// TwinCAT 3 PLC project Main
// ProgramVersion: 3.1.4024.0
// libraries:
//   Tc2_Standard, * (Beckhoff Automation GmbH)
//   Tc2_System, * (Beckhoff Automation GmbH)
//   Tc2_Utilities, * (Beckhoff Automation GmbH)
//   Tc3_DynamicMemory, * (Beckhoff Automation GmbH)
//   Tc3_JsonXml, * (Beckhoff Automation GmbH)
//   Tc3_Module, * (Beckhoff Automation GmbH)
//   TcUnit, * (www.tcunit.org)
//   mobject-core,0.4.0,mobject
// project tree:
//   mobject-collections/ MobjectCollectionsExample.TcPOU, MobjectCollectionsUnitTests.TcPOU
//   mobject-collections/Tests/ DictionaryForwardEnumerator_TestSuite.TcPOU (not stored), DictionaryKeyValueForwardEnumerator_TestSuite.TcPOU, Dictionary_TestSuite.TcPOU, LinkedListForwardEnumerator_TestSuite.TcPOU (not stored), LinkedList_TestSuite.TcPOU (not stored), OrderedDicKeyValueForwardEnumerator_TestSuite.TcPOU (not stored), OrderedDictionaryForwardEnumerator_TestSuite.TcPOU, OrderedDictionary_TestSuite.TcPOU, QueueForwardEnumerator_TestSuite.TcPOU (not stored), Queue_TestSuite.TcPOU, StackForwardEnumerator_TestSuite.TcPOU, Stack_TestSuite.TcPOU (not stored)
//   mobject-collections/Tests/Mocks/EventHandlers/ CollectionChangedEventHandler.TcPOU (not stored), CollectionDisposedEventHandler.TcPOU, CollectionEventHandler.TcPOU, CollectionEventHandlerBase.TcPOU (not stored), KeyValueCollectionChangedEventHandler.TcPOU, KeyValueCollectionDisposedEventHandler.TcPOU (not stored), KeyValueCollectionEventHandler.TcPOU (not stored)
//   mobject-converters/ MobjectConvertersUnitTests.TcPOU (not stored)
//   mobject-converters/Tests/ BOOL_TO_TestSuite.TcPOU, BYTE_TO_TestSuite.TcPOU (not stored), DATE_TO_TestSuite.TcPOU (not stored), DINT_TO_TestSuite.TcPOU (not stored), DT_TO_TestSuite.TcPOU, DWORD_TO_TestSuite.TcPOU, INT_TO_TestSuite.TcPOU (not stored), LINT_TO_TestSuite.TcPOU (not stored), LREAL_TO_TestSuite.TcPOU (not stored), LWORD_TO_TestSuite.TcPOU (not stored), REAL_TO_TestSuite.TcPOU (not stored), SINT_TO_TestSuite.TcPOU, STRING_TO_TestSuite.TcPOU (not stored), TIME_TO_TestSuite.TcPOU (not stored), TOD_TO_TestSuite.TcPOU (not stored), UDINT_TO_TestSuite.TcPOU (not stored), UINT_TO_TestSuite.TcPOU, ULINT_TO_TestSuite.TcPOU (not stored), USINT_TO_TestSuite.TcPOU (not stored), WORD_TO_TestSuite.TcPOU
//   mobject-datatypes/ MobjectDatatypesUnitTests.TcPOU
//   mobject-datatypes/Tests/ AliasDatatype_TestSuite.TcPOU, Datatype_TestSuite.TcPOU, EnumDatatype_TestSuite.TcPOU (not stored), StructuredDatatype_TestSuite.TcPOU, _ArrayDatatype_1D_TestSuite.TcPOU (not stored), _ArrayDatatype_2D_TestSuite.TcPOU, _ArrayDatatype_3D_TestSuite.TcPOU (not stored), _BIT_UsingMockStructure_TestSuite.TcPOU (not stored), _BOOL_TestSuite.TcPOU, _BYTE_TestSuite.TcPOU, _DINT_TestSuite.TcPOU (not stored), _DT_TestSuite.TcPOU, _DWORD_TestSuite.TcPOU, _INT_TestSuite.TcPOU, _LINT_TestSuite.TcPOU (not stored), _LREAL_TestSuite.TcPOU, _LWORD_TestSuite.TcPOU, _REAL_TestSuite.TcPOU (not stored), _SINT_TestSuite.TcPOU (not stored), _STRING_TestSuite.TcPOU, _TIME_OF_DAY_TestSuite.TcPOU, _TOD_TestSuite.TcPOU, _UDINT_TestSuite.TcPOU (not stored), _UINT_TestSuite.TcPOU (not stored), _ULINT_TestSuite.TcPOU (not stored), _USINT_TestSuite.TcPOU, _WORD_TestSuite.TcPOU
//   mobject-datatypes/Tests/Mocks/1DimArray/ _Array0to10OfBool.TcPOU
//   mobject-datatypes/Tests/Mocks/2DimArray/ _Array0to1_0to2OfBool.TcPOU
//   mobject-datatypes/Tests/Mocks/3DimArray/ _Array0to1_0to2_0to3OfBool.TcPOU
//   mobject-datatypes/Tests/Mocks/DUT/ MyStruct.TcDUT (not stored)
//   mobject-datatypes/Tests/Mocks/ MockAliasDatatype_HRESULT.TcPOU, MockDatatype_BOOL.TcPOU, MockEnumDatatype_E_TcEventClass.TcPOU, MockStructuredDatatype_TIMESTRUCT.TcPOU, _MyStruct.TcPOU
//   mobject-deserialization/ MobjectDeserializationUnitTests.TcPOU
//   mobject-deserialization/Tests/ CustomDeserializationFailedError_TestSuite.TcPOU (not stored), DeserializationErrorFactory_TestSuite.TcPOU (not stored), DeserializerGarbageCollector_TestSuite.TcPOU, IncorrectKeyTypeDeserializationError_TestSuite.TcPOU (not stored), IncorrectTypeDeserializationError_TestSuite.TcPOU (not stored), InvalidKeyDeserializationError_TestSuite.TcPOU (not stored), MissingKeyDeserializationError_TestSuite.TcPOU, InvalidArrayIndexDeserializationError_TestSuite.TcPOU
//   mobject-deserialization/Tests/Mocks/ MockDisposableDeserializer.TcPOU
//   mobject-disposable/ MobjectDisposableUnitTests.TcPOU (not stored)
//   mobject-disposable/Tests/ Disposable_TestSuite.TcPOU (not stored)
//   mobject-disposable/Tests/Mocks/ MockDisposable.TcPOU (not stored)
//   mobject-errors/ MobjectErrorsUnitTests.TcPOU (not stored)
//   mobject-errors/Tests/ Error_TestSuite.TcPOU, NullError_TestSuite.TcPOU
//   mobject-events/ MobjectEventsUnitTests.TcPOU (not stored)
//   mobject-events/Tests/ EventEmitterInterface_TestSuite.TcPOU, EventEmitter_TestSuite.TcPOU, EventHandlerInterface_TestSuite.TcPOU, EventTargetInterface_TestSuite.TcPOU (not stored)
//   mobject-events/Tests/Mocks/ MockEvent.TcPOU, MockEventHandler.TcPOU
//   mobject-json/ MobjectJsonUnitTests.TcPOU (not stored)
//   mobject-json/Tests/ JsonDeserializerArrayForwardEnumerator_TestSuite.TcPOU (not stored), JsonDeserializerObjectForwardEnumerator_TestSuite.TcPOU, JsonDeserializer_TestSuite.TcPOU, JsonDomParser_TestSuite.TcPOU (not stored), JsonSerializer_TestSuite.TcPOU
//   mobject-json/Tests/Mocks/ MockDeserializableUserObject.TcPOU (not stored), MockSerializableArray.TcPOU, MockSerializableUserObject.TcPOU (not stored)
//   / PlcTask.TcTTO (not stored)
//   Main/ MAIN.TcPOU
//   SharedMocks/ MockError.TcPOU (not stored), MockErrorVisitor.TcPOU, MockJsonSerializer.TcPOU (not stored)
// real-time tasks:
//   TASK PlcTask: cycle T#10ms, priority 20, ADS port 350

// ---- mobject-collections/MobjectCollectionsExample.TcPOU
PROGRAM MobjectCollectionsExample
VAR
END_VAR

END_PROGRAM

// ---- mobject-collections/MobjectCollectionsUnitTests.TcPOU
PROGRAM MobjectCollectionsUnitTests
VAR
	dictionary_TestSuite : Dictionary_TestSuite;
	dictionaryForwardEnumerator_TestSuite : DictionaryForwardEnumerator_TestSuite;
	dictionaryKeyValueForwardEnumerator_TestSuite : DictionaryKeyValueForwardEnumerator_TestSuite;
	orderedDictionary_TestSuite : OrderedDictionary_TestSuite;
	orderedDictionaryForwardEnumerator_TestSuite : OrderedDictionaryForwardEnumerator_TestSuite;
	orderedDicKeyValueForwardEnumerator_TestSuite : OrderedDicKeyValueForwardEnumerator_TestSuite;
    linkedList_TestSuite : LinkedList_TestSuite;
	linkedListForwardEnumerator_TestSuite : LinkedListForwardEnumerator_TestSuite;
    list_TestSuite : List_TestSuite;
    listEnumerator_TestSuite : ListForwardEnumerator_TestSuite;
	queue_TestSuite : Queue_TestSuite;
	queueForwardEnumerator_TestSuite : QueueForwardEnumerator_TestSuite;
    stack_TestSuite : Stack_TestSuite;
	stackForwardEnumerator_TestSuite : StackForwardEnumerator_TestSuite;
END_VAR

END_PROGRAM

// ---- mobject-collections/Tests/Dictionary_TestSuite.TcPOU
FUNCTION_BLOCK Dictionary_TestSuite EXTENDS TcUnit.FB_TestSuite
VAR
END_VAR

CheckAddOrUpdateCorrectlyAddsNewKey();
CheckAddOrUpdateCorrectlyUpdatesExistingKey();
CheckClear();
CheckContainsKeyIsFalse();
CheckContainsKeyIsTrue();
CheckCount();
CheckEnumeratorIsInvalidAfterChange();
CheckGetEnumerator();
CheckGetKeysReturnsACollection();
CheckGetKeysReturnsACollectionOfValidKeys();
CheckOffEvent();
CheckOnceEvent();
CheckOnChangedEvent();
CheckOnDisposedEvent();
CheckRemoveExisting();
CheckRemoveNonExisting();
CheckTryAddCorrectlyAddsNewKey();
CheckTryAddCorrectlyIgnoresUpdateWhenDuplicateFound();
CheckTryAddCorrectlyReturnsFalseWhenDuplicateFound();
CheckTryAddCorrectlyReturnsTrueWhenAddNewKey();
CheckTryGetValueTo();
CheckTryGetValue();
CheckWorksWithArrays();
CheckWorksWithIntegers();
CheckWorksWithStrings();
CheckIsEmptyWhenEmpty();
CheckIsEmptyWhenFull();

METHOD PUBLIC CheckAddOrUpdateCorrectlyAddsNewKey
VAR
	in : INT := 123;
	out : INT;
	expected : INT := 123;
	dictionary : Dictionary;
END_VAR
TEST('CheckAddOrUpdateCorrectlyAddsNewKey');

dictionary.AddOrUpdate('a',in);
dictionary.TryGetValue('a',out);

AssertEquals(
	Expected := expected,
	Actual := out,
	Message := 'Did not produce the expected result'
);

TEST_FINISHED();
END_METHOD

METHOD PUBLIC CheckAddOrUpdateCorrectlyUpdatesExistingKey
VAR
	in1 : INT := 123;
	in2 : INT := 456;
	out : INT;
	expected : INT := 456;
	dictionary : Dictionary;
END_VAR
TEST('CheckAddOrUpdateCorrectlyUpdatesExistingKey');

dictionary.AddOrUpdate('a',in1);
dictionary.AddOrUpdate('a',in2);
dictionary.TryGetValue('a',out);

AssertEquals(
	Expected := expected,
	Actual := out,
	Message := 'Did not produce the expected result'
);

TEST_FINISHED();
END_METHOD

METHOD PUBLIC CheckClear
VAR
	in1 : INT := 123;
	in2 : INT := 456;
	out : INT;
	expected : INT := 456;
	dictionary : Dictionary;
END_VAR
TEST('CheckClear');

dictionary.TryAdd('a',in1);
dictionary.Clear();
dictionary.TryAdd('a',in2); // if the dictionary was not empty then this would fail.
dictionary.TryGetValue('a',out);

// @TEST-ASSSERT
AssertEquals(
	Expected := expected,
	Actual := out,
	Message := 'Did not produce the expected result'
);

TEST_FINISHED();
END_METHOD

METHOD PUBLIC CheckContainsKeyIsFalse
VAR
	in1 : INT := 123;
	in2 : INT := 456;
	in3 : INT := 789;
	result : BOOL;
	dictionary : Dictionary;
END_VAR
TEST('CheckContainsKeyIsFalse');

dictionary.TryAdd('a',in1);
dictionary.TryAdd('b',in2);
dictionary.TryAdd('c',in3);

result := dictionary.ContainsKey('d');

AssertFalse(
	Condition := result,
	Message := 'Did not produce the expected result'
);

TEST_FINISHED();
END_METHOD

METHOD PUBLIC CheckContainsKeyIsTrue
VAR
	in1 : INT := 123;
	in2 : INT := 456;
	in3 : INT := 789;
	result : BOOL;
	dictionary : Dictionary;
END_VAR
TEST('CheckContainsKeyIsTrue');

dictionary.TryAdd('a',in1);
dictionary.TryAdd('b',in2);
dictionary.TryAdd('c',in3);

result := dictionary.ContainsKey('b');

AssertTrue(
	Condition := result,
	Message := 'Did not produce the expected result'
);

TEST_FINISHED();
END_METHOD

METHOD PUBLIC CheckCount
VAR
	in1 : INT := 123;
	in2 : INT := 456;
	in3 : INT := 789;
	out : DINT;
	expected : DINT := 3;
	dictionary : Dictionary;
END_VAR
TEST('CheckCount');

dictionary.TryAdd('a',in1);
dictionary.TryAdd('b',in2);
dictionary.TryAdd('c',in3);
out := dictionary.Count;

AssertEquals(
	Expected := expected,
	Actual := out,
	Message := 'Did not produce the expected result'
);

TEST_FINISHED();
END_METHOD

METHOD PUBLIC CheckEnumeratorIsInvalidAfterChange
VAR
	in : INT := 123;
	result : BOOL;
	dictionary : Dictionary;
	enumerator : I_ForwardEnumerator;
END_VAR
TEST('CheckEnumeratorIsInvalidAfterChange');

enumerator := dictionary.GetEnumerator();
dictionary.TryAdd('a',in);

result := enumerator.IsValid;
enumerator.Dispose();

AssertFalse(
	Condition := result,
	Message := 'Method returned true'
);

TEST_FINISHED();
END_METHOD

METHOD PUBLIC CheckGetEnumerator
VAR
	enumerator : I_ForwardEnumerator;
	dictionary : Dictionary;
END_VAR
TEST('CheckGetEnumerator');

enumerator := dictionary.GetEnumerator();

AssertTrue(
	Condition := (enumerator <> 0),
	Message := 'Did not return an enumerator'
);

enumerator.Dispose();

TEST_FINISHED();
END_METHOD

METHOD PUBLIC CheckGetKeysReturnsACollection
VAR
	result : BOOL;
	dictionary : Dictionary;
	collection : I_Collection;
END_VAR
TEST('CheckGetKeysReturnsACollection');

collection := dictionary.GetKeys();

result := collection <> 0;

IF result THEN
	collection.Dispose();
END_IF

AssertTrue(
	Condition := result,
	Message := 'Did not produce the expected result'
);

TEST_FINISHED();
END_METHOD

METHOD PUBLIC CheckGetKeysReturnsACollectionOfValidKeys
VAR
	in1 : INT := 123;
	in2 : INT := 456;
	in3 : INT := 789;
	out : ARRAY [0..2] OF T_MAXSTRING;
	expected : ARRAY [0..2] OF T_MAXSTRING;
	result,resulta,resultb,resultc : BOOL;
	dictionary : Dictionary;
	collection : I_Collection;
END_VAR
TEST('CheckGetKeysReturnsACollectionOfValidKeys');

// clear the out and expected variables as strings may contain left over data
memset(ADR(out),0,SIZEOF(out));
memset(ADR(expected),0,SIZEOF(expected));

// now create the "expected"
expected[0] := 'a';
expected[1] := 'b';
expected[2] := 'c';

// now setup the test
dictionary.TryAdd('a',in1);
dictionary.TryAdd('b',in2);
dictionary.TryAdd('c',in3);

collection := dictionary.GetKeys();
collection.TryCopyTo(out);
collection.Dispose();

// create the test result
resulta := expected[0] = out[0];
resultb := expected[1] = out[1];
resultc := expected[2] = out[2];
result := resulta AND resultb AND resultc;

AssertTrue(
	Condition := result,
	Message := 'Did not return an enumerator'
);

TEST_FINISHED();
END_METHOD

METHOD PUBLIC CheckIsEmptyWhenEmpty
VAR
	result : BOOL;
	dictionary : Dictionary;
END_VAR
TEST('CheckIsEmptyWhenEmpty');

// @TEST-RUN
result := dictionary.IsEmpty;

// @TEST-ASSSERT
AssertTrue(
	Condition := result,
	Message := 'Incorrect state of IsEmpty'
);

TEST_FINISHED();
END_METHOD

METHOD PUBLIC CheckIsEmptyWhenFull
VAR
	in : INT := 123;
	result : BOOL;
	dictionary : Dictionary;
END_VAR
TEST('CheckIsEmptyWhenFull');

// @TEST-FIXTURE
dictionary.AddOrUpdate('a',in);

// @TEST-RUN
result := dictionary.IsEmpty;

// @TEST-ASSSERT
AssertFalse(
	Condition := result,
	Message := 'Incorrect state of IsEmpty'
);

TEST_FINISHED();
END_METHOD

METHOD PUBLIC CheckOffEvent
VAR
	value : INT := 123;
	dictionary : Dictionary;
	handler : KeyValueCollectionChangedEventHandler(ExpectedOriginator := dictionary);
END_VAR
TEST('CheckOffEvent');

dictionary.OnEvent('OnChanged',handler);
dictionary.OffEvent('OnChanged',handler);

dictionary.TryAdd('a',value);

AssertFalse(
	Condition := handler.EventReceived,
	Message := 'OnceEvent emitted the OnChanged event more than once'
);

TEST_FINISHED();
END_METHOD

METHOD PUBLIC CheckOnceEvent
VAR
	value : INT := 123;
	dictionary : Dictionary;
	handler : KeyValueCollectionChangedEventHandler(ExpectedOriginator := dictionary);
END_VAR
TEST('CheckOnceEvent');

dictionary.OnceEvent('OnChanged',handler);
dictionary.TryAdd('a',value);
handler.Reset();

dictionary.TryAdd('a',value);

AssertFalse(
	Condition := handler.EventReceived,
	Message := 'OnceEvent emitted the OnChanged event more than once'
);

TEST_FINISHED();
END_METHOD

METHOD PUBLIC CheckOnChangedEvent
VAR
	value : INT := 123;
	dictionary : Dictionary;
	handler : KeyValueCollectionChangedEventHandler(ExpectedOriginator := dictionary);
END_VAR
TEST('CheckOnChangedEvent');

dictionary.OnEvent('OnChanged', handler);
dictionary.TryAdd('a',value);

AssertTrue(
	Condition := handler.EventReceived,
	Message := 'Did not emit the OnChanged event'
);

AssertTrue(
	Condition := handler.FromExpectedOriginator,
	Message := 'Did not include itself in the OnChanged event'
);

TEST_FINISHED();
END_METHOD

METHOD PUBLIC CheckOnDisposedEvent
VAR
	value : INT := 123;
	pDictionary : POINTER TO Dictionary;
	handler : KeyValueCollectionDisposedEventHandler(ExpectedOriginator := 0);
END_VAR
TEST('CheckOnDisposedEvent');

pDictionary := __NEW(Dictionary);
handler.SetExpectedOriginator(pDictionary^);
pDictionary^.OnEvent('OnDisposed', handler);

pDictionary^.Dispose();

AssertTrue(
	Condition := handler.EventReceived,
	Message := 'Did not emit the OnDisposed event'
);

AssertTrue(
	Condition := handler.FromExpectedOriginator,
	Message := 'Did not include itself in the OnDisposed event'
);

TEST_FINISHED();
END_METHOD

METHOD PRIVATE CheckRemoveExisting
VAR
	in1 : INT := 123;
	in2 : INT := 456;
	in3 : INT := 789;
	result : BOOL;
	dictionary : Dictionary;
END_VAR
TEST('CheckRemoveExisting');

dictionary.TryAdd('a',in1);
dictionary.TryAdd('b',in2);
dictionary.TryAdd('c',in3);

dictionary.Remove('c');

result := dictionary.ContainsKey('c');

AssertFalse(
	Condition := result,
	Message := 'Did not produce the expected result'
);

TEST_FINISHED();
END_METHOD

METHOD PRIVATE CheckRemoveNonExisting
VAR
	in1 : INT := 123;
	in2 : INT := 456;
	in3 : INT := 789;
	out : DINT;
	expected : DINT := 3;
	dictionary : Dictionary;
END_VAR
TEST('CheckRemoveNonExisting');

dictionary.TryAdd('a',in1);
dictionary.TryAdd('b',in2);
dictionary.TryAdd('c',in3);

dictionary.Remove('d');

out := dictionary.Count;

AssertEquals(
	Expected := expected,
	Actual := out,
	Message := 'Did not produce the expected result'
);

TEST_FINISHED();
END_METHOD

METHOD PUBLIC CheckTryAddCorrectlyAddsNewKey
VAR
	in : INT := 123;
	out : INT;
	expected : INT := 123;
	dictionary : Dictionary;
END_VAR
TEST('CheckTryAddCorrectlyAddsNewKey');

dictionary.TryAdd('a',in);
dictionary.TryGetValue('a',out);

AssertEquals(
	Expected := expected,
	Actual := out,
	Message := 'Did not produce the expected result'
);

TEST_FINISHED();
END_METHOD

METHOD PUBLIC CheckTryAddCorrectlyIgnoresUpdateWhenDuplicateFound
VAR
	in1 : INT := 123;
	in2 : INT := 456;
	out : INT;
	expected : INT := 123;
	result : BOOL;
	dictionary : Dictionary;
END_VAR
TEST('CheckTryAddCorrectlyIgnoresUpdateWhenDuplicateFound');

dictionary.TryAdd('a',in1);
dictionary.TryAdd('a',in2);
dictionary.TryGetValue('a',out);

AssertEquals(
	Expected := expected,
	Actual := out,
	Message := 'Did not produce the expected result'
);

TEST_FINISHED();
END_METHOD

METHOD PUBLIC CheckTryAddCorrectlyReturnsFalseWhenDuplicateFound
VAR
	in1 : INT := 123;
	in2 : INT := 456;
	result : BOOL;
	dictionary : Dictionary;
END_VAR
TEST('CheckTryAddCorrectlyReturnsFalseWhenDuplicateFound');

dictionary.TryAdd('a',in1);
result := dictionary.TryAdd('a',in2);

AssertFalse(
	Condition := result,
	Message := 'Did not produce the expected result'
);

TEST_FINISHED();
END_METHOD

METHOD PUBLIC CheckTryAddCorrectlyReturnsTrueWhenAddNewKey
VAR
	in : INT := 123;
	result : BOOL;
	dictionary : Dictionary;
END_VAR
TEST('CheckTryAddCorrectlyReturnsTrueWhenAddNewKey');

result := dictionary.TryAdd('a',in);

AssertTrue(
	Condition := result,
	Message := 'Did not produce the expected result'
);

TEST_FINISHED();
END_METHOD

METHOD PUBLIC CheckTryGetValue
VAR
	in : INT := 123;
	out : INT;
	expected : INT := 123;
	dictionary : Dictionary;
END_VAR
TEST('CheckTryGetValue');

dictionary.AddOrUpdate('a',in);
dictionary.TryGetValue('a',out);

AssertEquals(
	Expected := expected,
	Actual := out,
	Message := 'Did not produce the expected result'
);

TEST_FINISHED();
END_METHOD

METHOD PUBLIC CheckTryGetValueTo
VAR
	in : INT := 123;
	out : INT;
	expected : INT := 123;
	dictionary : Dictionary;
END_VAR
TEST('CheckTryGetValueTo');

dictionary.AddOrUpdate('a',in);
dictionary.TryGetValueTo('a',ADR(out),SIZEOF(out));

AssertEquals(
	Expected := expected,
	Actual := out,
	Message := 'Did not produce the expected result'
);

TEST_FINISHED();
END_METHOD

METHOD PUBLIC CheckWorksWithArrays
VAR
	in : ARRAY [0..1] OF REAL := [0.1,2.3];
	out : ARRAY [0..1] OF REAL;
	expected : ARRAY [0..1] OF REAL := [0.1,2.3];
	dictionary : Dictionary;
END_VAR
TEST('CheckWorksWithArrays');

dictionary.TryAdd('a',in);
dictionary.TryGetValue('a',out);

AssertEquals(
	Expected := expected,
	Actual := out,
	Message := 'Did not produce the expected result'
);

TEST_FINISHED();
END_METHOD

METHOD PUBLIC CheckWorksWithIntegers
VAR
	in : INT := 123;
	out : INT;
	expected : INT := 123;
	dictionary : Dictionary;
END_VAR
TEST('CheckWorksWithIntegers');

dictionary.TryAdd('a',in);
dictionary.TryGetValue('a',out);

AssertEquals(
	Expected := expected,
	Actual := out,
	Message := 'Did not produce the expected result'
);

TEST_FINISHED();
END_METHOD

METHOD PUBLIC CheckWorksWithStrings
VAR
	in : STRING := 'test';
	out : STRING;
	expected : STRING := 'test';
	dictionary : Dictionary;
END_VAR
TEST('CheckWorksWithStrings');

dictionary.TryAdd('a',in);
dictionary.TryGetValue('a',out);

AssertEquals(
	Expected := expected,
	Actual := out,
	Message := 'Did not produce the expected result'
);

TEST_FINISHED();
END_METHOD

END_FUNCTION_BLOCK

// ---- mobject-collections/Tests/Mocks/EventHandlers/KeyValueCollectionChangedEventHandler.TcPOU
FUNCTION_BLOCK KeyValueCollectionChangedEventHandler EXTENDS KeyValueCollectionEventHandler

METHOD PUBLIC HandleEvent
VAR_INPUT
	Event : I_Event;
END_VAR
VAR
	changedEvent : I_KeyValueCollectionChangedEvent;
END_VAR
IF __QUERYINTERFACE(Event, changedEvent) THEN
	_eventReceived := TRUE;
	fromExpected := changedEvent.Target = expectedOriginator;
END_IF
END_METHOD

END_FUNCTION_BLOCK

// ---- mobject-collections/Tests/DictionaryKeyValueForwardEnumerator_TestSuite.TcPOU
FUNCTION_BLOCK DictionaryKeyValueForwardEnumerator_TestSuite EXTENDS TcUnit.FB_TestSuite
VAR
END_VAR

CheckIsValidAtStart();
CheckKey();
CheckMoveNextReturnsFalseAtTheEnd();
CheckMoveNextReturnsTrueSingleItem();
CheckMoveNextReturnsFalseWhenEmpty();
CheckMoveNextReturnsTrueMultipleItems();
CheckReset();
CheckTryGet();
CheckTryGetTo();
CheckWorksWithArrays();
CheckWorksWithIntegers();
CheckWorksWithStrings();

METHOD PRIVATE CheckIsValidAtStart
VAR
	result : BOOL;
	dictionary : Dictionary;
	enumerator : I_KeyValueForwardEnumerator;
END_VAR
TEST('CheckIsValidAtStart');

enumerator := dictionary.GetKeyValueEnumerator();

result := enumerator.IsValid;
enumerator.Dispose();

AssertTrue(
	Condition := result,
	Message := 'IsValid returned false'
);

TEST_FINISHED();
END_METHOD

METHOD PRIVATE CheckKey
VAR
	in1 : STRING := 'test1';
	in2 : STRING := 'test2';
	in3 : STRING := 'test3';
	out1 : STRING;
	out2 : STRING;
	out3 : STRING;
	expected1 : STRING := 'a';
	expected2 : STRING := 'b';
	expected3 : STRING := 'c';
	dictionary : Dictionary;
	enumerator : I_KeyValueForwardEnumerator;
END_VAR
TEST('CheckKey');

dictionary.TryAdd('a',in1);
dictionary.TryAdd('b',in2);
dictionary.TryAdd('c',in3);

enumerator := dictionary.GetKeyValueEnumerator();

enumerator.MoveNext();
out1 := enumerator.Key;
enumerator.MoveNext();
out2 := enumerator.Key;
enumerator.MoveNext();
out3 := enumerator.Key;

enumerator.Dispose();

AssertEquals(
	Expected := expected1,
	Actual := out1,
	Message := 'Did not produce the expected 1st key'
);

AssertEquals(
	Expected := expected2,
	Actual := out2,
	Message := 'Did not produce the expected 2nd key'
);

AssertEquals(
	Expected := expected3,
	Actual := out3,
	Message := 'Did not produce the expected 3rd key'
);

TEST_FINISHED();
END_METHOD

METHOD PRIVATE CheckMoveNextReturnsFalseAtTheEnd
VAR
	in1 : INT := 123;
	result : BOOL;
	dictionary : Dictionary;
	enumerator : I_KeyValueForwardEnumerator;
END_VAR
TEST('CheckMoveNextReturnsFalseAtTheEnd');

dictionary.TryAdd('a',in1);
enumerator := dictionary.GetKeyValueEnumerator();

enumerator.MoveNext();
result := enumerator.MoveNext();

enumerator.Dispose();

AssertFalse(result,
    'MoveNext did not correctly signal the end of the enumeration');
	
TEST_FINISHED();
END_METHOD

METHOD PRIVATE CheckMoveNextReturnsFalseWhenEmpty
VAR
	result : BOOL;
	dictionary : Dictionary;
	enumerator : I_KeyValueForwardEnumerator;
	count : DINT;
END_VAR
TEST('CheckMoveNextReturnsFalseWhenEmpty');

count := dictionary.Count;
enumerator := dictionary.GetKeyValueEnumerator();

result := enumerator.MoveNext();
enumerator.Dispose();

AssertFalse(Condition := result,
    Message := 'MoveNext did not correctly signal the end of the enumeration');

TEST_FINISHED();
END_METHOD

METHOD PRIVATE CheckMoveNextReturnsTrueMultipleItems
VAR
	in1 : INT := 123;
	in2 : INT := 456;
	in3 : INT := 789;
	result : BOOL;
	dictionary : Dictionary;
	enumerator : I_KeyValueForwardEnumerator;
END_VAR
TEST('CheckMoveNextReturnsTrueMultipleItems');

dictionary.TryAdd('a',in1);
dictionary.TryAdd('b',in2);
dictionary.TryAdd('c',in3);
enumerator := dictionary.GetKeyValueEnumerator();

result := enumerator.MoveNext();
enumerator.Dispose();

AssertTrue(result, 'MoveNext did not correctly signal there were more items to follow');

TEST_FINISHED();
END_METHOD

METHOD PRIVATE CheckMoveNextReturnsTrueSingleItem
VAR
	in1 : INT := 123;
	result : BOOL;
	dictionary : Dictionary;
	enumerator : I_KeyValueForwardEnumerator;
END_VAR
TEST('CheckMoveNextReturnsTrueSingleItem');

dictionary.TryAdd('a',in1);
enumerator := dictionary.GetKeyValueEnumerator();

result := enumerator.MoveNext();
enumerator.Dispose();

AssertTrue(result,
    'MoveNext did not correctly signal there were more items to follow');
	
TEST_FINISHED();
END_METHOD

METHOD PRIVATE CheckReset
VAR
	in1 : ARRAY [0..1] OF REAL := [0.1,2.3];
	in2 : ARRAY [0..1] OF REAL := [1.2,3.4];
	in3 : ARRAY [0..1] OF REAL := [2.3,4.5];
	out : ARRAY [0..1] OF REAL;
	expected : ARRAY [0..1] OF REAL := [0.1,2.3];
	dictionary : Dictionary;
	enumerator : I_KeyValueForwardEnumerator;
END_VAR
TEST('CheckReset');

dictionary.TryAdd('a',in1);
dictionary.TryAdd('b',in2);
dictionary.TryAdd('c',in3);

enumerator := dictionary.GetKeyValueEnumerator();

enumerator.MoveNext();
enumerator.MoveNext();
enumerator.Reset();
enumerator.MoveNext();
enumerator.TryGet(out);

enumerator.Dispose();

AssertEquals(
	Expected := expected,
	Actual := out,
	Message := 'Did not produce the expected result'
);

TEST_FINISHED();
END_METHOD

METHOD PRIVATE CheckTryGet
VAR
	in : INT := 123;
	out : INT;
	expected : INT := 123;
	result : BOOL;
	dictionary : Dictionary;
	enumerator : I_KeyValueForwardEnumerator;
END_VAR
TEST('CheckTryGet');

dictionary.TryAdd('a',in);
enumerator := dictionary.GetKeyValueEnumerator();
enumerator.MoveNext();

result := enumerator.TryGet(out);
enumerator.Dispose();

AssertTrue(
	Condition := result,
	Message := 'Method returned false'
);

AssertEquals(
	Expected := expected,
	Actual := out,
	Message := 'Did not produce the expected result'
);

TEST_FINISHED();
END_METHOD

METHOD PRIVATE CheckTryGetTo
VAR
	in : INT := 123;
	out : INT;
	expected : INT := 123;
	result : BOOL;
	dictionary : Dictionary;
	enumerator : I_KeyValueForwardEnumerator;
END_VAR
TEST('CheckTryGetTo');

dictionary.TryAdd('a',in);
enumerator := dictionary.GetKeyValueEnumerator();
enumerator.MoveNext();

result := enumerator.TryGetTo(ADR(out),SIZEOF(out));
enumerator.Dispose();

AssertTrue(
	Condition := result,
	Message := 'Method returned false'
);

AssertEquals(
	Expected := expected,
	Actual := out,
	Message := 'Did not produce the expected result'
);

TEST_FINISHED();
END_METHOD

METHOD PRIVATE CheckWorksWithArrays
VAR
	in1 : ARRAY [0..1] OF REAL := [0.1,2.3];
	in2 : ARRAY [0..1] OF REAL := [1.2,3.4];
	in3 : ARRAY [0..1] OF REAL := [2.3,4.5];
	out1 : ARRAY [0..1] OF REAL;
	out2 : ARRAY [0..1] OF REAL;
	out3 : ARRAY [0..1] OF REAL;
	expected1 : ARRAY [0..1] OF REAL := [0.1,2.3];
	expected2 : ARRAY [0..1] OF REAL := [1.2,3.4];
	expected3 : ARRAY [0..1] OF REAL := [2.3,4.5];
	dictionary : Dictionary;
	enumerator : I_KeyValueForwardEnumerator;
END_VAR
TEST('CheckWorksWithArrays');

dictionary.TryAdd('c',in3);
dictionary.TryAdd('b',in2);
dictionary.TryAdd('a',in1);

enumerator := dictionary.GetKeyValueEnumerator();

enumerator.MoveNext();
enumerator.TryGet(out1);
enumerator.MoveNext();
enumerator.TryGet(out2);
enumerator.MoveNext();
enumerator.TryGet(out3);

enumerator.Dispose();

AssertEquals(
	Expected := expected1,
	Actual := out1,
	Message := 'Did not produce the expected 1st result'
);

AssertEquals(
	Expected := expected2,
	Actual := out2,
	Message := 'Did not produce the expected 2nd result'
);

AssertEquals(
	Expected := expected3,
	Actual := out3,
	Message := 'Did not produce the expected 3rd result'
);

TEST_FINISHED();
END_METHOD

METHOD PRIVATE CheckWorksWithIntegers
VAR
	in1 : INT := 123;
	in2 : INT := 234;
	in3 : INT := 345;
	out1 : INT;
	out2 : INT;
	out3 : INT;
	expected1 : INT := 123;
	expected2 : INT := 234;
	expected3 : INT := 345;
	dictionary : Dictionary;
	enumerator : I_KeyValueForwardEnumerator;
END_VAR
TEST('CheckWorksWithIntegers');

dictionary.TryAdd('c',in3);
dictionary.TryAdd('b',in2);
dictionary.TryAdd('a',in1);

enumerator := dictionary.GetKeyValueEnumerator();

enumerator.MoveNext();
enumerator.TryGet(out1);
enumerator.MoveNext();
enumerator.TryGet(out2);
enumerator.MoveNext();
enumerator.TryGet(out3);

enumerator.Dispose();

AssertEquals(
	Expected := expected1,
	Actual := out1,
	Message := 'Did not produce the expected 1st result'
);

AssertEquals(
	Expected := expected2,
	Actual := out2,
	Message := 'Did not produce the expected 2nd result'
);

AssertEquals(
	Expected := expected3,
	Actual := out3,
	Message := 'Did not produce the expected 3rd result'
);

TEST_FINISHED();
END_METHOD

METHOD PRIVATE CheckWorksWithStrings
VAR
	in1 : STRING := 'test1';
	in2 : STRING := 'test2';
	in3 : STRING := 'test3';
	out1 : STRING;
	out2 : STRING;
	out3 : STRING;
	expected1 : STRING := 'test1';
	expected2 : STRING := 'test2';
	expected3 : STRING := 'test3';
	dictionary : Dictionary;
	enumerator : I_KeyValueForwardEnumerator;
END_VAR
TEST('CheckWorksWithStrings');

dictionary.TryAdd('c',in3);
dictionary.TryAdd('b',in2);
dictionary.TryAdd('a',in1);

enumerator := dictionary.GetKeyValueEnumerator();

enumerator.MoveNext();
enumerator.TryGet(out1);
enumerator.MoveNext();
enumerator.TryGet(out2);
enumerator.MoveNext();
enumerator.TryGet(out3);

enumerator.Dispose();

AssertEquals(
	Expected := expected1,
	Actual := out1,
	Message := 'Did not produce the expected 1st result'
);

AssertEquals(
	Expected := expected2,
	Actual := out2,
	Message := 'Did not produce the expected 2nd result'
);

AssertEquals(
	Expected := expected3,
	Actual := out3,
	Message := 'Did not produce the expected 3rd result'
);

TEST_FINISHED();
END_METHOD

END_FUNCTION_BLOCK

// ---- mobject-collections/Tests/OrderedDictionary_TestSuite.TcPOU
FUNCTION_BLOCK OrderedDictionary_TestSuite EXTENDS TcUnit.FB_TestSuite
VAR
END_VAR

CheckAddOrUpdateCorrectlyAddsNewKey();
CheckAddOrUpdateCorrectlyUpdatesExistingKey();
CheckClear();
CheckContainsKeyIsFalse();
CheckContainsKeyIsTrue();
CheckCount();
CheckEnumeratorIsInvalidAfterChange();
CheckGetEnumerator();
CheckGetKeysReturnsACollection();
CheckGetKeysReturnsACollectionOfValidKeys();
CheckOffEvent();
CheckOnceEvent();
CheckOnChangedEvent();
CheckOnDisposedEvent();
CheckRemoveExisting();
CheckRemoveNonExisting();
CheckTryAddCorrectlyAddsNewKey();
CheckTryAddCorrectlyIgnoresUpdateWhenDuplicateFound();
CheckTryAddCorrectlyReturnsFalseWhenDuplicateFound();
CheckTryAddCorrectlyReturnsTrueWhenAddNewKey();
CheckTryGetValueTo();
CheckTryGetValue();
CheckWorksWithArrays();
CheckWorksWithIntegers();
CheckWorksWithManyItems();
CheckWorksWithStrings();
CheckIsEmptyWhenEmpty();
CheckIsEmptyWhenFull();

METHOD PUBLIC CheckAddOrUpdateCorrectlyAddsNewKey
VAR
	in : INT := 123;
	out : INT;
	expected : INT := 123;
	dictionary : OrderedDictionary;
END_VAR
TEST('CheckAddOrUpdateCorrectlyAddsNewKey');

dictionary.AddOrUpdate('a',in);
dictionary.TryGetValue('a',out);

AssertEquals(
	Expected := expected,
	Actual := out,
	Message := 'Did not produce the expected result'
);

TEST_FINISHED();
END_METHOD

METHOD PUBLIC CheckAddOrUpdateCorrectlyUpdatesExistingKey
VAR
	in1 : INT := 123;
	in2 : INT := 456;
	out : INT;
	expected : INT := 456;
	dictionary : OrderedDictionary;
END_VAR
TEST('CheckAddOrUpdateCorrectlyUpdatesExistingKey');

dictionary.AddOrUpdate('a',in1);
dictionary.AddOrUpdate('a',in2);
dictionary.TryGetValue('a',out);

AssertEquals(
	Expected := expected,
	Actual := out,
	Message := 'Did not produce the expected result'
);

TEST_FINISHED();
END_METHOD

METHOD PUBLIC CheckClear
VAR
	in1 : INT := 123;
	in2 : INT := 456;
	out : INT;
	expected : INT := 456;
	dictionary : OrderedDictionary;
END_VAR
TEST('CheckClear');

dictionary.TryAdd('a',in1);
dictionary.Clear();
dictionary.TryAdd('a',in2); // if the dictionary was not empty then this would fail.
dictionary.TryGetValue('a',out);

// @TEST-ASSSERT
AssertEquals(
	Expected := expected,
	Actual := out,
	Message := 'Did not produce the expected result'
);

TEST_FINISHED();
END_METHOD

METHOD PUBLIC CheckContainsKeyIsFalse
VAR
	in1 : INT := 123;
	in2 : INT := 456;
	in3 : INT := 789;
	result : BOOL;
	dictionary : OrderedDictionary;
END_VAR
TEST('CheckContainsKeyIsFalse');

dictionary.TryAdd('a',in1);
dictionary.TryAdd('b',in2);
dictionary.TryAdd('c',in3);

result := dictionary.ContainsKey('d');

AssertFalse(
	Condition := result,
	Message := 'Did not produce the expected result'
);

TEST_FINISHED();
END_METHOD

METHOD PUBLIC CheckContainsKeyIsTrue
VAR
	in1 : INT := 123;
	in2 : INT := 456;
	in3 : INT := 789;
	result : BOOL;
	dictionary : OrderedDictionary;
END_VAR
TEST('CheckContainsKeyIsTrue');

dictionary.TryAdd('a',in1);
dictionary.TryAdd('b',in2);
dictionary.TryAdd('c',in3);

result := dictionary.ContainsKey('b');

AssertTrue(
	Condition := result,
	Message := 'Did not produce the expected result'
);

TEST_FINISHED();
END_METHOD

METHOD PUBLIC CheckCount
VAR
	in1 : INT := 123;
	in2 : INT := 456;
	in3 : INT := 789;
	out : DINT;
	expected : DINT := 3;
	dictionary : OrderedDictionary;
END_VAR
TEST('CheckCount');

dictionary.TryAdd('a',in1);
dictionary.TryAdd('b',in2);
dictionary.TryAdd('c',in3);
out := dictionary.Count;

AssertEquals(
	Expected := expected,
	Actual := out,
	Message := 'Did not produce the expected result'
);

TEST_FINISHED();
END_METHOD

METHOD PUBLIC CheckEnumeratorIsInvalidAfterChange
VAR
	in : INT := 123;
	result : BOOL;
	dictionary : OrderedDictionary;
	enumerator : I_ForwardEnumerator;
END_VAR
TEST('CheckEnumeratorIsInvalidAfterChange');

enumerator := dictionary.GetEnumerator();
dictionary.TryAdd('a',in);

result := enumerator.IsValid;
enumerator.Dispose();

AssertFalse(
	Condition := result,
	Message := 'Method returned true'
);

TEST_FINISHED();
END_METHOD

METHOD PUBLIC CheckGetEnumerator
VAR
	enumerator : I_ForwardEnumerator;
	dictionary : OrderedDictionary;
END_VAR
TEST('CheckGetEnumerator');

enumerator := dictionary.GetEnumerator();

AssertTrue(
	Condition := (enumerator <> 0),
	Message := 'Did not return an enumerator'
);

enumerator.Dispose();

TEST_FINISHED();
END_METHOD

METHOD PUBLIC CheckGetKeysReturnsACollection
VAR
	result : BOOL;
	dictionary : OrderedDictionary;
	collection : I_Collection;
END_VAR
TEST('CheckGetKeysReturnsACollection');

collection := dictionary.GetKeys();

result := collection <> 0;

IF result THEN
	collection.Dispose();
END_IF

AssertTrue(
	Condition := result,
	Message := 'Did not produce the expected result'
);

TEST_FINISHED();
END_METHOD

METHOD PUBLIC CheckGetKeysReturnsACollectionOfValidKeys
VAR
	in1 : INT := 123;
	in2 : INT := 456;
	in3 : INT := 789;
	out : ARRAY [0..2] OF T_MAXSTRING;
	expected : ARRAY [0..2] OF T_MAXSTRING;
	result,resulta,resultb,resultc : BOOL;
	dictionary : OrderedDictionary;
	collection : I_Collection;
END_VAR
TEST('CheckGetKeysReturnsACollectionOfValidKeys');

// clear the out and expected variables as strings may contain left over data
memset(ADR(out),0,SIZEOF(out));
memset(ADR(expected),0,SIZEOF(expected));

// now create the "expected"
expected[0] := 'a';
expected[1] := 'b';
expected[2] := 'c';

// now setup the test
dictionary.TryAdd('a',in1);
dictionary.TryAdd('b',in2);
dictionary.TryAdd('c',in3);

collection := dictionary.GetKeys();
collection.TryCopyTo(out);
collection.Dispose();

// create the test result
resulta := expected[0] = out[0];
resultb := expected[1] = out[1];
resultc := expected[2] = out[2];
result := resulta AND resultb AND resultc;

AssertTrue(
	Condition := result,
	Message := 'Did not return an enumerator'
);

TEST_FINISHED();
END_METHOD

METHOD PUBLIC CheckIsEmptyWhenEmpty
VAR
	result : BOOL;
	dictionary : OrderedDictionary;
END_VAR
TEST('CheckIsEmptyWhenEmpty');

// @TEST-RUN
result := dictionary.IsEmpty;

// @TEST-ASSSERT
AssertTrue(
	Condition := result,
	Message := 'Incorrect state of IsEmpty'
);

TEST_FINISHED();
END_METHOD

METHOD PUBLIC CheckIsEmptyWhenFull
VAR
	in : INT := 123;
	result : BOOL;
	dictionary : OrderedDictionary;
END_VAR
TEST('CheckIsEmptyWhenFull');

// @TEST-FIXTURE
dictionary.AddOrUpdate('a',in);

// @TEST-RUN
result := dictionary.IsEmpty;

// @TEST-ASSSERT
AssertFalse(
	Condition := result,
	Message := 'Incorrect state of IsEmpty'
);

TEST_FINISHED();
END_METHOD

METHOD PUBLIC CheckOffEvent
VAR
	value : INT := 123;
	dictionary : OrderedDictionary;
	handler : KeyValueCollectionChangedEventHandler(ExpectedOriginator := dictionary);
END_VAR
TEST('CheckOffEvent');

dictionary.OnEvent('OnChanged',handler);
dictionary.OffEvent('OnChanged',handler);

dictionary.TryAdd('a',value);

AssertFalse(
	Condition := handler.EventReceived,
	Message := 'OnceEvent emitted the OnChanged event more than once'
);

TEST_FINISHED();
END_METHOD

METHOD PUBLIC CheckOnceEvent
VAR
	value : INT := 123;
	dictionary : OrderedDictionary;
	handler : KeyValueCollectionChangedEventHandler(ExpectedOriginator := dictionary);
END_VAR
TEST('CheckOnceEvent');

dictionary.OnceEvent('OnChanged',handler);
dictionary.TryAdd('a',value);
handler.Reset();

dictionary.TryAdd('a',value);

AssertFalse(
	Condition := handler.EventReceived,
	Message := 'OnceEvent emitted the OnChanged event more than once'
);

TEST_FINISHED();
END_METHOD

METHOD PUBLIC CheckOnChangedEvent
VAR
	value : INT := 123;
	dictionary : OrderedDictionary;
	handler : KeyValueCollectionChangedEventHandler(ExpectedOriginator := dictionary);
END_VAR
TEST('CheckOnChangedEvent');

dictionary.OnEvent('OnChanged', handler);
dictionary.TryAdd('a',value);

AssertTrue(
	Condition := handler.EventReceived,
	Message := 'Did not emit the OnChanged event'
);

AssertTrue(
	Condition := handler.FromExpectedOriginator,
	Message := 'Did not include itself in the OnChanged event'
);

TEST_FINISHED();
END_METHOD

METHOD PUBLIC CheckOnDisposedEvent
VAR
	value : INT := 123;
	pDictionary : POINTER TO OrderedDictionary;
	handler : KeyValueCollectionDisposedEventHandler(ExpectedOriginator := 0);
END_VAR
TEST('CheckOnDisposedEvent');

pDictionary := __NEW(OrderedDictionary);
handler.SetExpectedOriginator(pDictionary^);
pDictionary^.OnEvent('OnDisposed', handler);

pDictionary^.Dispose();

AssertTrue(
	Condition := handler.EventReceived,
	Message := 'Did not emit the OnDisposed event'
);

AssertTrue(
	Condition := handler.FromExpectedOriginator,
	Message := 'Did not include itself in the OnDisposed event'
);

TEST_FINISHED();
END_METHOD

METHOD PRIVATE CheckRemoveExisting
VAR
	in1 : INT := 123;
	in2 : INT := 456;
	in3 : INT := 789;
	result : BOOL;
	dictionary : OrderedDictionary;
END_VAR
TEST('CheckRemoveExisting');

dictionary.TryAdd('a',in1);
dictionary.TryAdd('b',in2);
dictionary.TryAdd('c',in3);

dictionary.Remove('c');

result := dictionary.ContainsKey('c');

AssertFalse(
	Condition := result,
	Message := 'Did not produce the expected result'
);

TEST_FINISHED();
END_METHOD

METHOD PRIVATE CheckRemoveNonExisting
VAR
	in1 : INT := 123;
	in2 : INT := 456;
	in3 : INT := 789;
	out : DINT;
	expected : DINT := 3;
	dictionary : OrderedDictionary;
END_VAR
TEST('CheckRemoveNonExisting');

dictionary.TryAdd('a',in1);
dictionary.TryAdd('b',in2);
dictionary.TryAdd('c',in3);

dictionary.Remove('d');

out := dictionary.Count;

AssertEquals(
	Expected := expected,
	Actual := out,
	Message := 'Did not produce the expected result'
);

TEST_FINISHED();
END_METHOD

METHOD PUBLIC CheckTryAddCorrectlyAddsNewKey
VAR
	in : INT := 123;
	out : INT;
	expected : INT := 123;
	dictionary : OrderedDictionary;
END_VAR
TEST('CheckTryAddCorrectlyAddsNewKey');

dictionary.TryAdd('a',in);
dictionary.TryGetValue('a',out);

AssertEquals(
	Expected := expected,
	Actual := out,
	Message := 'Did not produce the expected result'
);

TEST_FINISHED();
END_METHOD

METHOD PUBLIC CheckTryAddCorrectlyIgnoresUpdateWhenDuplicateFound
VAR
	in1 : INT := 123;
	in2 : INT := 456;
	out : INT;
	expected : INT := 123;
	result : BOOL;
	dictionary : OrderedDictionary;
END_VAR
TEST('CheckTryAddCorrectlyIgnoresUpdateWhenDuplicateFound');

dictionary.TryAdd('a',in1);
dictionary.TryAdd('a',in2);
dictionary.TryGetValue('a',out);

AssertEquals(
	Expected := expected,
	Actual := out,
	Message := 'Did not produce the expected result'
);

TEST_FINISHED();
END_METHOD

METHOD PUBLIC CheckTryAddCorrectlyReturnsFalseWhenDuplicateFound
VAR
	in1 : INT := 123;
	in2 : INT := 456;
	result : BOOL;
	dictionary : OrderedDictionary;
END_VAR
TEST('CheckTryAddCorrectlyReturnsFalseWhenDuplicateFound');

dictionary.TryAdd('a',in1);
result := dictionary.TryAdd('a',in2);

AssertFalse(
	Condition := result,
	Message := 'Did not produce the expected result'
);

TEST_FINISHED();
END_METHOD

METHOD PUBLIC CheckTryAddCorrectlyReturnsTrueWhenAddNewKey
VAR
	in : INT := 123;
	result : BOOL;
	dictionary : OrderedDictionary;
END_VAR
TEST('CheckTryAddCorrectlyReturnsTrueWhenAddNewKey');

result := dictionary.TryAdd('a',in);

AssertTrue(
	Condition := result,
	Message := 'Did not produce the expected result'
);

TEST_FINISHED();
END_METHOD

METHOD PUBLIC CheckTryGetValue
VAR
	in : INT := 123;
	out : INT;
	expected : INT := 123;
	dictionary : OrderedDictionary;
END_VAR
TEST('CheckTryGetValue');

dictionary.AddOrUpdate('a',in);
dictionary.TryGetValue('a',out);

AssertEquals(
	Expected := expected,
	Actual := out,
	Message := 'Did not produce the expected result'
);

TEST_FINISHED();
END_METHOD

METHOD PUBLIC CheckTryGetValueTo
VAR
	in : INT := 123;
	out : INT;
	expected : INT := 123;
	dictionary : OrderedDictionary;
END_VAR
TEST('CheckTryGetValueTo');

dictionary.AddOrUpdate('a',in);
dictionary.TryGetValueTo('a',ADR(out),SIZEOF(out));

AssertEquals(
	Expected := expected,
	Actual := out,
	Message := 'Did not produce the expected result'
);

TEST_FINISHED();
END_METHOD

METHOD PUBLIC CheckWorksWithArrays
VAR
	in : ARRAY [0..1] OF REAL := [0.1,2.3];
	out : ARRAY [0..1] OF REAL;
	expected : ARRAY [0..1] OF REAL := [0.1,2.3];
	dictionary : OrderedDictionary;
END_VAR
TEST('CheckWorksWithArrays');

dictionary.TryAdd('a',in);
dictionary.TryGetValue('a',out);

AssertEquals(
	Expected := expected,
	Actual := out,
	Message := 'Did not produce the expected result'
);

TEST_FINISHED();
END_METHOD

METHOD PUBLIC CheckWorksWithIntegers
VAR
	in : INT := 123;
	out : INT;
	expected : INT := 123;
	dictionary : OrderedDictionary;
END_VAR
TEST('CheckWorksWithIntegers');

dictionary.TryAdd('a',in);
dictionary.TryGetValue('a',out);

AssertEquals(
	Expected := expected,
	Actual := out,
	Message := 'Did not produce the expected result'
);

TEST_FINISHED();
END_METHOD

METHOD PUBLIC CheckWorksWithManyItems
VAR
	in : INT := 0;
	out : DINT;
	expected : DINT := 13;
	dictionary : OrderedDictionary;
END_VAR
TEST('CheckWorksWithManyItems');

dictionary.TryAdd('TCVN_PPM_NONE', in);
dictionary.TryAdd('TCVN_PPM_MONO1P', in);
dictionary.TryAdd('TCVN_PPM_MONO2P', in);
dictionary.TryAdd('TCVN_PPM_MONO4P', in);
dictionary.TryAdd('TCVN_PPM_MONO10PACKED', in);
dictionary.TryAdd('TCVN_PPM_MONO12PACKED', in);
dictionary.TryAdd('TCVN_PPM_RGB10V1PACKED', in);
dictionary.TryAdd('TCVN_PPM_RGB10P32', in);
dictionary.TryAdd('TCVN_PPM_RGB12V1PACKED', in);
dictionary.TryAdd('TCVN_PPM_RGB565P', in);
dictionary.TryAdd('TCVN_PPM_BGR565P', in);
dictionary.TryAdd('TCVN_PPM_MONO10P', in);
dictionary.TryAdd('TCVN_PPM_MONO12P', in);

out := dictionary.Count;

dictionary.Clear();

AssertEquals(
	Expected := expected,
	Actual := out,
	Message := 'Did not produce the expected count when adding many items'
);

TEST_FINISHED();
END_METHOD

METHOD PUBLIC CheckWorksWithStrings
VAR
	in : STRING := 'test';
	out : STRING;
	expected : STRING := 'test';
	dictionary : OrderedDictionary;
END_VAR
TEST('CheckWorksWithStrings');

dictionary.TryAdd('a',in);
dictionary.TryGetValue('a',out);

AssertEquals(
	Expected := expected,
	Actual := out,
	Message := 'Did not produce the expected result'
);

TEST_FINISHED();
END_METHOD

END_FUNCTION_BLOCK

// ---- mobject-collections/Tests/OrderedDictionaryForwardEnumerator_TestSuite.TcPOU
FUNCTION_BLOCK OrderedDictionaryForwardEnumerator_TestSuite EXTENDS TcUnit.FB_TestSuite
VAR
END_VAR

CheckIsValidAtStart();
CheckMoveNextReturnsFalseAtTheEnd();
CheckMoveNextReturnsTrueSingleItem();
CheckMoveNextReturnsFalseWhenEmpty();
CheckMoveNextReturnsTrueMultipleItems();
CheckReset();
CheckTryGet();
CheckTryGetTo();
CheckWorksWithArrays();
CheckWorksWithIntegers();
CheckWorksWithStrings();

METHOD PRIVATE CheckIsValidAtStart
VAR
	result : BOOL;
	dictionary : OrderedDictionary;
	enumerator : I_ForwardEnumerator;
END_VAR
TEST('CheckIsValidAtStart');

enumerator := dictionary.GetEnumerator();

result := enumerator.IsValid;
enumerator.Dispose();

AssertTrue(
	Condition := result,
	Message := 'IsValid returned false'
);

TEST_FINISHED();
END_METHOD

METHOD PRIVATE CheckMoveNextReturnsFalseAtTheEnd
VAR
	in1 : INT := 123;
	result : BOOL;
	dictionary : OrderedDictionary;
	enumerator : I_ForwardEnumerator;
END_VAR
TEST('CheckMoveNextReturnsFalseAtTheEnd');

dictionary.TryAdd('a',in1);
enumerator := dictionary.GetEnumerator();

enumerator.MoveNext();
result := enumerator.MoveNext();

enumerator.Dispose();

AssertFalse(result,
    'MoveNext did not correctly signal the end of the enumeration');
	
TEST_FINISHED();
END_METHOD

METHOD PRIVATE CheckMoveNextReturnsFalseWhenEmpty
VAR
	result : BOOL;
	dictionary : OrderedDictionary;
	enumerator : I_ForwardEnumerator;
	count : DINT;
END_VAR
TEST('CheckMoveNextReturnsFalseWhenEmpty');

count := dictionary.Count;
enumerator := dictionary.GetEnumerator();

result := enumerator.MoveNext();
enumerator.Dispose();

AssertFalse(Condition := result,
    Message := 'MoveNext did not correctly signal the end of the enumeration');

TEST_FINISHED();
END_METHOD

METHOD PRIVATE CheckMoveNextReturnsTrueMultipleItems
VAR
	in1 : INT := 123;
	in2 : INT := 456;
	in3 : INT := 789;
	result : BOOL;
	dictionary : OrderedDictionary;
	enumerator : I_ForwardEnumerator;
END_VAR
TEST('CheckMoveNextReturnsTrueMultipleItems');

dictionary.TryAdd('a',in1);
dictionary.TryAdd('b',in2);
dictionary.TryAdd('c',in3);
enumerator := dictionary.GetEnumerator();

result := enumerator.MoveNext();
enumerator.Dispose();

AssertTrue(result, 'MoveNext did not correctly signal there were more items to follow');

TEST_FINISHED();
END_METHOD

METHOD PRIVATE CheckMoveNextReturnsTrueSingleItem
VAR
	in1 : INT := 123;
	result : BOOL;
	dictionary : OrderedDictionary;
	enumerator : I_ForwardEnumerator;
END_VAR
TEST('CheckMoveNextReturnsTrueSingleItem');

dictionary.TryAdd('a',in1);
enumerator := dictionary.GetEnumerator();

result := enumerator.MoveNext();
enumerator.Dispose();

AssertTrue(result,
    'MoveNext did not correctly signal there were more items to follow');
	
TEST_FINISHED();
END_METHOD

METHOD PRIVATE CheckReset
VAR
	in1 : ARRAY [0..1] OF REAL := [0.1,2.3];
	in2 : ARRAY [0..1] OF REAL := [1.2,3.4];
	in3 : ARRAY [0..1] OF REAL := [2.3,4.5];
	out : ARRAY [0..1] OF REAL;
	expected : ARRAY [0..1] OF REAL := [0.1,2.3];
	dictionary : OrderedDictionary;
	enumerator : I_ForwardEnumerator;
END_VAR
TEST('CheckReset');

dictionary.TryAdd('a',in1);
dictionary.TryAdd('b',in2);
dictionary.TryAdd('c',in3);

enumerator := dictionary.GetEnumerator();

enumerator.MoveNext();
enumerator.MoveNext();
enumerator.Reset();
enumerator.MoveNext();
enumerator.TryGet(out);

enumerator.Dispose();

AssertEquals(
	Expected := expected,
	Actual := out,
	Message := 'Did not produce the expected result'
);

TEST_FINISHED();
END_METHOD

METHOD PRIVATE CheckTryGet
VAR
	in : INT := 123;
	out : INT;
	expected : INT := 123;
	result : BOOL;
	dictionary : OrderedDictionary;
	enumerator : I_ForwardEnumerator;
END_VAR
TEST('CheckTryGet');

dictionary.TryAdd('a',in);
enumerator := dictionary.GetEnumerator();
enumerator.MoveNext();

result := enumerator.TryGet(out);
enumerator.Dispose();

AssertTrue(
	Condition := result,
	Message := 'Method returned false'
);

AssertEquals(
	Expected := expected,
	Actual := out,
	Message := 'Did not produce the expected result'
);

TEST_FINISHED();
END_METHOD

METHOD PRIVATE CheckTryGetTo
VAR
	in : INT := 123;
	out : INT;
	expected : INT := 123;
	result : BOOL;
	dictionary : OrderedDictionary;
	enumerator : I_ForwardEnumerator;
END_VAR
TEST('CheckTryGetTo');

dictionary.TryAdd('a',in);
enumerator := dictionary.GetEnumerator();
enumerator.MoveNext();

result := enumerator.TryGetTo(ADR(out),SIZEOF(out));
enumerator.Dispose();

AssertTrue(
	Condition := result,
	Message := 'Method returned false'
);

AssertEquals(
	Expected := expected,
	Actual := out,
	Message := 'Did not produce the expected result'
);

TEST_FINISHED();
END_METHOD

METHOD PRIVATE CheckWorksWithArrays
VAR
	in1 : ARRAY [0..1] OF REAL := [0.1,2.3];
	in2 : ARRAY [0..1] OF REAL := [1.2,3.4];
	in3 : ARRAY [0..1] OF REAL := [2.3,4.5];
	out1 : ARRAY [0..1] OF REAL;
	out2 : ARRAY [0..1] OF REAL;
	out3 : ARRAY [0..1] OF REAL;
	expected1 : ARRAY [0..1] OF REAL := [0.1,2.3];
	expected2 : ARRAY [0..1] OF REAL := [1.2,3.4];
	expected3 : ARRAY [0..1] OF REAL := [2.3,4.5];
	dictionary : OrderedDictionary;
	enumerator : I_ForwardEnumerator;
END_VAR
TEST('CheckWorksWithArrays');

dictionary.TryAdd('c',in1);
dictionary.TryAdd('b',in2);
dictionary.TryAdd('a',in3);

enumerator := dictionary.GetEnumerator();

enumerator.MoveNext();
enumerator.TryGet(out1);
enumerator.MoveNext();
enumerator.TryGet(out2);
enumerator.MoveNext();
enumerator.TryGet(out3);

enumerator.Dispose();

AssertEquals(
	Expected := expected1,
	Actual := out1,
	Message := 'Did not produce the expected 1st result'
);

AssertEquals(
	Expected := expected2,
	Actual := out2,
	Message := 'Did not produce the expected 2nd result'
);

AssertEquals(
	Expected := expected3,
	Actual := out3,
	Message := 'Did not produce the expected 3rd result'
);

TEST_FINISHED();
END_METHOD

METHOD PRIVATE CheckWorksWithIntegers
VAR
	in1 : INT := 123;
	in2 : INT := 234;
	in3 : INT := 345;
	out1 : INT;
	out2 : INT;
	out3 : INT;
	expected1 : INT := 123;
	expected2 : INT := 234;
	expected3 : INT := 345;
	dictionary : OrderedDictionary;
	enumerator : I_ForwardEnumerator;
END_VAR
TEST('CheckWorksWithIntegers');

dictionary.TryAdd('c',in1);
dictionary.TryAdd('b',in2);
dictionary.TryAdd('a',in3);

enumerator := dictionary.GetEnumerator();

enumerator.MoveNext();
enumerator.TryGet(out1);
enumerator.MoveNext();
enumerator.TryGet(out2);
enumerator.MoveNext();
enumerator.TryGet(out3);

enumerator.Dispose();

AssertEquals(
	Expected := expected1,
	Actual := out1,
	Message := 'Did not produce the expected 1st result'
);

AssertEquals(
	Expected := expected2,
	Actual := out2,
	Message := 'Did not produce the expected 2nd result'
);

AssertEquals(
	Expected := expected3,
	Actual := out3,
	Message := 'Did not produce the expected 3rd result'
);

TEST_FINISHED();
END_METHOD

METHOD PRIVATE CheckWorksWithStrings
VAR
	in1 : STRING := 'test1';
	in2 : STRING := 'test2';
	in3 : STRING := 'test3';
	out1 : STRING;
	out2 : STRING;
	out3 : STRING;
	expected1 : STRING := 'test1';
	expected2 : STRING := 'test2';
	expected3 : STRING := 'test3';
	dictionary : OrderedDictionary;
	enumerator : I_ForwardEnumerator;
END_VAR
TEST('CheckWorksWithStrings');

dictionary.TryAdd('c',in1);
dictionary.TryAdd('b',in2);
dictionary.TryAdd('a',in3);

enumerator := dictionary.GetEnumerator();

enumerator.MoveNext();
enumerator.TryGet(out1);
enumerator.MoveNext();
enumerator.TryGet(out2);
enumerator.MoveNext();
enumerator.TryGet(out3);

enumerator.Dispose();

AssertEquals(
	Expected := expected1,
	Actual := out1,
	Message := 'Did not produce the expected 1st result'
);

AssertEquals(
	Expected := expected2,
	Actual := out2,
	Message := 'Did not produce the expected 2nd result'
);

AssertEquals(
	Expected := expected3,
	Actual := out3,
	Message := 'Did not produce the expected 3rd result'
);

TEST_FINISHED();
END_METHOD

END_FUNCTION_BLOCK

// ---- mobject-collections/Tests/Queue_TestSuite.TcPOU
FUNCTION_BLOCK PUBLIC Queue_TestSuite EXTENDS TcUnit.FB_TestSuite

// check datatypes are handled correctly
CheckListWorksWithIntegers();
CheckListWorksWithStrings();
CheckListWorksWithArrays();

// all other checks
CheckQueueImplementsI_Queue();
CheckContains();
CheckClear();
CheckCount();
CheckAddItem();
CheckTryRemoveItem();
CheckTryDequeueRemovesTheItem();
CheckTryDequeueReturnsTheCorrectValue();
CheckTryPeekReturnsTheCorrectValue();
CheckTryPeekDoesNotRemoveTheItem();
CheckOnChangedEvent();
CheckOnDisposedEvent();
CheckOnceEvent();
CheckOffEvent();
CheckTryCopyTo();
CheckTryCopyToLocation();
CheckQueueOrderIsCorrect();
CheckListReturnsEnumerator();
CheckEnumeratorIsInvalidAfterChange();
CheckIsEmptyWhenEmpty();
CheckIsEmptyWhenFull();

METHOD PUBLIC CheckAddItem
VAR
	in1 : INT := 123;
	in2 : INT := 456;
	in3 : INT := 789;
	result : BOOL;
	queue : Queue;
END_VAR
TEST('CheckAddItem');

// @TEST-FIXTURE
queue.Enqueue(in1); // (lifo->) 123
queue.Enqueue(in2); // (lifo->) 123, 456

// @TEST-RUN
queue.AddItem(in3); // (lifo->) 123, 456, 789
result := queue.Contains(in3);

// @TEST-ASSSERT
AssertTrue(
	Condition := result,
	Message := 'Method returned false'
);

TEST_FINISHED();
END_METHOD

METHOD PUBLIC CheckClear
VAR
	in1 : INT := 123;
	in2 : INT := 456;
	in3 : INT := 789;
	queue : Queue;
END_VAR
TEST('CheckClear');

// @TEST-FIXTURE
queue.Enqueue(in1); // (lifo->) 123
queue.Enqueue(in2); // (lifo->) 123, 456
queue.Enqueue(in2); // (lifo->) 123, 456, 789

// @TEST-RUN
queue.Clear();

// @TEST-ASSSERT
AssertTrue(
	Condition := queue.Count = 0,
	Message := 'The count is not zero'
);

TEST_FINISHED();
END_METHOD

METHOD PUBLIC CheckContains
VAR
	in1 : INT := 123;
	in2 : INT := 456;
	in3 : INT := 789;
	result : BOOL;
	queue : Queue;
END_VAR
TEST('CheckContains');

// @TEST-FIXTURE
queue.Enqueue(in1); // (lifo->) 123
queue.Enqueue(in2); // (lifo->) 123, 456
queue.Enqueue(in2); // (lifo->) 123, 456, 789

// @TEST-RUN
result := queue.Contains(in2);

// @TEST-ASSSERT
AssertTrue(
	Condition := result,
	Message := 'Did not find the item in the queue'
);

TEST_FINISHED();
END_METHOD

METHOD PUBLIC CheckCount
VAR
	in1 : INT := 123;
	in2 : INT := 456;
	in3 : INT := 789;
	total : DINT;
	expected : DINT := 3;
	queue : Queue;
END_VAR
TEST('CheckCount');

// @TEST-FIXTURE
queue.Enqueue(in1); // (lifo->) 123
queue.Enqueue(in2); // (lifo->) 123, 456
queue.Enqueue(in2); // (lifo->) 123, 456, 789

// @TEST-RUN
total := queue.Count;

// @TEST-ASSSERT
AssertEquals(
	Expected := expected,
	Actual := total,
	Message := 'Incorrect count'
);

TEST_FINISHED();
END_METHOD

METHOD PUBLIC CheckEnumeratorIsInvalidAfterChange
VAR
	in : INT := 123;
	result : BOOL;
	queue : Queue;
	enumerator : I_ForwardEnumerator;
END_VAR
TEST('CheckEnumeratorIsInvalidAfterChange');

// @TEST-FIXTURE
enumerator := queue.GetEnumerator();
queue.Enqueue(in);

// @TEST-RUN
result := enumerator.IsValid;
enumerator.Dispose();

// @TEST-ASSSERT
AssertFalse(
	Condition := result,
	Message := 'Method returned true'
);

TEST_FINISHED();
END_METHOD

METHOD PUBLIC CheckIsEmptyWhenEmpty
VAR
	result : BOOL;
	queue : Queue;
END_VAR
TEST('CheckIsEmptyWhenEmpty');

// @TEST-RUN
result := queue.IsEmpty;

// @TEST-ASSSERT
AssertTrue(
	Condition := result,
	Message := 'Incorrect state of IsEmpty'
);

TEST_FINISHED();
END_METHOD

METHOD PUBLIC CheckIsEmptyWhenFull
VAR
	in : INT := 123;
	result : BOOL;
	queue : Queue;
END_VAR
TEST('CheckIsEmptyWhenFull');

// @TEST-FIXTURE
queue.Enqueue(in);

// @TEST-RUN
result := queue.IsEmpty;

// @TEST-ASSSERT
AssertFalse(
	Condition := result,
	Message := 'Incorrect state of IsEmpty'
);

TEST_FINISHED();
END_METHOD

METHOD PUBLIC CheckListReturnsEnumerator
VAR
	in1 : INT := 123;
	in2 : INT := 456;
	in3 : INT := 789;
	enumerator : I_ForwardEnumerator;
	queue : Queue;
END_VAR
TEST('CheckListReturnsEnumerator');

// @TEST-FIXTURE
queue.Enqueue(in1); // (lifo->) 123
queue.Enqueue(in2); // (lifo->) 123, 456
queue.Enqueue(in2); // (lifo->) 123, 456, 789

// @TEST-RUN
enumerator := queue.GetEnumerator();

// @TEST-ASSSERT
AssertTrue(
	Condition := (enumerator <> 0),
	Message := 'Did not return an enumerator'
);

// @TEST-DISPOSE
enumerator.Dispose();

TEST_FINISHED();
END_METHOD

METHOD PUBLIC CheckListWorksWithArrays
VAR
	in : ARRAY [0..1] OF REAL := [0.1,2.3];
	out : ARRAY [0..1] OF REAL;
	expected : ARRAY [0..1] OF REAL := [0.1,2.3];
	result : BOOL;
	queue : Queue;
END_VAR
TEST('CheckListWorksWithArrays');

// @TEST-FIXTURE
queue.Enqueue(in);

// @TEST-RUN
result := queue.TryDequeue(out);

// @TEST-ASSSERT
AssertTrue(
	Condition := result,
	Message := 'Method returned false'
);

AssertEquals(
	Expected := expected,
	Actual := out,
	Message := 'Did not produce the expected result'
);

TEST_FINISHED();
END_METHOD

METHOD PUBLIC CheckListWorksWithIntegers
VAR
	in : INT := 123;
	out : INT;
	expected : INT := 123;
	result : BOOL;
	queue : Queue;
END_VAR
TEST('CheckListWorksWithIntegers');

// @TEST-FIXTURE
queue.Enqueue(in);

// @TEST-RUN
result := queue.TryDequeue(out);

// @TEST-ASSSERT
AssertTrue(
	Condition := result,
	Message := 'Method returned false'
);

AssertEquals(
	Expected := expected,
	Actual := out,
	Message := 'Did not produce the expected result'
);

TEST_FINISHED();
END_METHOD

METHOD PUBLIC CheckListWorksWithStrings
VAR
	in : STRING := 'test';
	out : STRING;
	expected : STRING := 'test';
	result : BOOL;
	queue : Queue;
END_VAR
TEST('CheckListWorksWithStrings');

// @TEST-FIXTURE
queue.Enqueue(in);

// @TEST-RUN
result := queue.TryDequeue(out);

// @TEST-ASSSERT
AssertTrue(
	Condition := result,
	Message := 'Method returned false'
);

AssertEquals(
	Expected := expected,
	Actual := out,
	Message := 'Did not produce the expected result'
);

TEST_FINISHED();
END_METHOD

METHOD PUBLIC CheckOffEvent
VAR
	value : INT := 123;
	queue : queue;
	handler : CollectionChangedEventHandler(ExpectedOriginator := queue);
END_VAR
TEST('CheckOffEvent');

// @TEST-FIXTURE
queue.OnEvent('OnChanged',handler);
queue.OffEvent('OnChanged',handler);

// @TEST-RUN
queue.Enqueue(value);

// @TEST-ASSSERT
AssertFalse(
	Condition := handler.EventReceived,
	Message := 'OnceEvent emitted the OnChanged event more than once'
);

TEST_FINISHED();
END_METHOD

METHOD PUBLIC CheckOnceEvent
VAR
	value : INT := 123;
	queue : Queue;
	handler : CollectionChangedEventHandler(ExpectedOriginator := queue);
END_VAR
TEST('CheckOnceEvent');

// @TEST-FIXTURE
queue.OnceEvent('OnChanged',handler);
queue.Enqueue(value);
handler.Reset();

// @TEST-RUN
queue.Enqueue(value);

// @TEST-ASSSERT
AssertFalse(
	Condition := handler.EventReceived,
	Message := 'OnceEvent emitted the OnChanged event more than once'
);

TEST_FINISHED();
END_METHOD

METHOD PUBLIC CheckOnChangedEvent
VAR
	value : INT := 123;
	queue : Queue;
	handler : CollectionChangedEventHandler(ExpectedOriginator := queue);
END_VAR
TEST('CheckOnChangedEvent');

// @TEST-FIXTURE
queue.OnEvent('OnChanged', handler);

// @TEST-RUN
queue.Enqueue(value);

// @TEST-ASSSERT
AssertTrue(
	Condition := handler.EventReceived,
	Message := 'Did not emit the OnChanged event'
);

AssertTrue(
	Condition := handler.FromExpectedOriginator,
	Message := 'Did not include itself in the OnChanged event'
);

TEST_FINISHED();
END_METHOD

METHOD PUBLIC CheckOnDisposedEvent
VAR
	value : INT := 123;
	pQueue : POINTER TO Queue;
	handler : CollectionDisposedEventHandler(ExpectedOriginator := 0);
END_VAR
TEST('CheckOnDisposedEvent');

// @TEST-FIXTURE
pQueue := __NEW(Queue);
handler.SetExpectedOriginator(pQueue^);
pQueue^.OnEvent('OnDisposed', handler);

// @TEST-RUN
pQueue^.Dispose();

// @TEST-ASSSERT
AssertTrue(
	Condition := handler.EventReceived,
	Message := 'Did not emit the OnDisposed event'
);

AssertTrue(
	Condition := handler.FromExpectedOriginator,
	Message := 'Did not include itself in the OnDisposed event'
);

TEST_FINISHED();
END_METHOD

METHOD PUBLIC CheckQueueImplementsI_Queue
VAR
	queue : Queue;
    iQueue : I_Queue := queue;
    result : BOOL;
END_VAR
TEST('CheckQueueImplementsI_Queue');

// @TEST-FIXTURE

// @TEST-RUN
result := iQueue <> 0;

// @TEST-ASSSERT
AssertTrue(
	Condition := result,
	Message := 'Did not implement I_Queue'
);

TEST_FINISHED();
END_METHOD

METHOD PUBLIC CheckQueueOrderIsCorrect
VAR
	in1 : INT := 123;
	in2 : INT := 456;
	in3 : INT := 789;
	out1, out2, out3 : INT;
	expected1 : INT := 123;
	expected2 : INT := 456;
	expected3 : INT := 789;
	result1, result2, result3 : BOOL;
	queue : Queue;
END_VAR
TEST('CheckQueueOrderIsCorrect');

// @TEST-FIXTURE
queue.Enqueue(in1); // (lifo->) 123
queue.Enqueue(in2); // (lifo->) 123, 456
queue.Enqueue(in3); // (lifo->) 123, 456, 789

// @TEST-RUN
result1 := queue.TryDequeue(out1); // (lifo->) 456, 789
result2 := queue.TryDequeue(out2); // (lifo->) 789
result3 := queue.TryDequeue(out3); // (lifo->) 

// @TEST-ASSSERT
AssertTrue(
	Condition := result1 AND result2 AND result3,
	Message := 'Method returned false'
);

AssertEquals(
	Expected := expected1,
	Actual := out1,
	Message := 'Did not produce the expected result'
);

AssertEquals(
	Expected := expected2,
	Actual := out2,
	Message := 'Did not produce the expected result'
);

AssertEquals(
	Expected := expected3,
	Actual := out3,
	Message := 'Did not produce the expected result'
);

TEST_FINISHED();
END_METHOD

METHOD PUBLIC CheckTryCopyTo
VAR
	in1 : INT := 123;
	in2 : INT := 456;
	in3 : INT := 789;
	out : ARRAY [0..2] OF INT;
	expected : ARRAY [0..2] OF INT := [123,456,789];
	queue : Queue;
END_VAR
TEST('CheckTryCopyTo');

// @TEST-FIXTURE
queue.Enqueue(in1); // (lifo->) 123
queue.Enqueue(in2); // (lifo->) 123, 456
queue.Enqueue(in3); // (lifo->) 123, 456, 789

// @TEST-RUN
queue.TryCopyTo(out);

// @TEST-ASSSERT
AssertEquals(
	Expected := expected,
	Actual := out,
	Message := 'Did not produce the expected result'
);

TEST_FINISHED();
END_METHOD

METHOD PUBLIC CheckTryCopyToLocation
VAR
	in1 : INT := 123;
	in2 : INT := 456;
	in3 : INT := 789;
	out : ARRAY [0..2] OF INT;
	expected : ARRAY [0..2] OF INT := [123,456,789];
	queue : Queue;
END_VAR
TEST('CheckTryCopyToLocation');

// @TEST-FIXTURE
queue.Enqueue(in1); // (lifo->) 123
queue.Enqueue(in2); // (lifo->) 123, 456
queue.Enqueue(in3); // (lifo->) 123, 456, 789

// @TEST-RUN
queue.TryCopyToLocation(ADR(out),SIZEOF(out));

// @TEST-ASSSERT
AssertEquals(
	Expected := expected,
	Actual := out,
	Message := 'Did not produce the expected result'
);

TEST_FINISHED();
END_METHOD

METHOD PUBLIC CheckTryDequeueRemovesTheItem
VAR
	in : INT := 123;
	out : INT;
	total : DINT;
	expected : DINT := 0;
	queue : Queue;
END_VAR
TEST('CheckTryDequeueDoesNotRemoveTheItem');

// @TEST-FIXTURE
queue.Enqueue(in); // (lifo->) 123

// @TEST-RUN
queue.TryDequeue(out);
total := queue.Count;

// @TEST-ASSSERT
AssertEquals(
	Expected := expected,
	Actual := total,
	Message := 'Incorrect count'
);

TEST_FINISHED();
END_METHOD

METHOD PUBLIC CheckTryDequeueReturnsTheCorrectValue
VAR
	in : INT := 123;
	out : INT;
	expected : INT := 123;
	result : BOOL;
	queue : Queue;
END_VAR
TEST('CheckTryDequeueReturnsTheCorrectValue');

// @TEST-FIXTURE
queue.Enqueue(in);

// @TEST-RUN
result := queue.TryPeek(out);

// @TEST-ASSSERT
AssertTrue(
	Condition := result,
	Message := 'Method returned false'
);

AssertEquals(
	Expected := expected,
	Actual := out,
	Message := 'Did not produce the expected result'
);

TEST_FINISHED();
END_METHOD

METHOD PUBLIC CheckTryPeekDoesNotRemoveTheItem
VAR
	in : INT := 123;
	out : INT;
	total : DINT;
	expected : DINT := 1;
	queue : Queue;
END_VAR
TEST('CheckTryPeekDoesNotRemoveTheItem');

// @TEST-FIXTURE
queue.Enqueue(in); // (lifo->) 123

// @TEST-RUN
queue.TryPeek(out);
total := queue.Count;

// @TEST-ASSSERT
AssertEquals(
	Expected := expected,
	Actual := total,
	Message := 'Incorrect count'
);

TEST_FINISHED();
END_METHOD

METHOD PUBLIC CheckTryPeekReturnsTheCorrectValue
VAR
	in : INT := 123;
	out : INT;
	expected : INT := 123;
	result : BOOL;
	queue : Queue;
END_VAR
TEST('CheckTryPeekReturnsTheCorrectValue');

// @TEST-FIXTURE
queue.Enqueue(in);

// @TEST-RUN
result := queue.TryPeek(out);

// @TEST-ASSSERT
AssertTrue(
	Condition := result,
	Message := 'Method returned false'
);

AssertEquals(
	Expected := expected,
	Actual := out,
	Message := 'Did not produce the expected result'
);

TEST_FINISHED();
END_METHOD

METHOD PUBLIC CheckTryRemoveItem
VAR
	in1 : INT := 123;
	in2 : INT := 456;
	in3 : INT := 789;
	result : BOOL;
	queue : Queue;
END_VAR
TEST('CheckTryRemoveItem');

// @TEST-FIXTURE
queue.Enqueue(in1); // (lifo->) 123
queue.Enqueue(in2); // (lifo->) 123, 456
queue.Enqueue(in3); // (lifo->) 123, 456, 789

// @TEST-RUN
queue.TryRemoveItem(in2); // (lifo->) 123, 789
result := queue.Contains(in2);

// @TEST-ASSSERT
AssertFalse(
	Condition := result,
	Message := 'Method returned true'
);

TEST_FINISHED();
END_METHOD

END_FUNCTION_BLOCK

// ---- mobject-collections/Tests/Mocks/EventHandlers/CollectionDisposedEventHandler.TcPOU
FUNCTION_BLOCK CollectionDisposedEventHandler EXTENDS CollectionEventHandler

METHOD PUBLIC HandleEvent
VAR_INPUT
	Event : I_Event;
END_VAR
VAR
	disposedEvent : I_CollectionDisposedEvent;
END_VAR
IF __QUERYINTERFACE(Event, disposedEvent) THEN
	_eventReceived := TRUE;
	fromExpected := disposedEvent.Target = expectedOriginator;
END_IF
END_METHOD

END_FUNCTION_BLOCK

// ---- mobject-collections/Tests/Mocks/EventHandlers/CollectionEventHandler.TcPOU
FUNCTION_BLOCK ABSTRACT CollectionEventHandler EXTENDS CollectionEventHandlerBase
VAR
	expectedOriginator : I_Collection;
END_VAR

METHOD FB_init : BOOL
VAR_INPUT
	bInitRetains : BOOL; // if TRUE, the retain variables are initialized (warm start / cold start)
	bInCopyCode : BOOL;  // if TRUE, the instance afterwards gets moved into the copy code (online change)
	ExpectedOriginator : I_Collection;
END_VAR
SetExpectedOriginator(ExpectedOriginator);
END_METHOD

METHOD PUBLIC SetExpectedOriginator
VAR_INPUT
	ExpectedOriginator : I_Collection;
END_VAR
THIS^.expectedOriginator := ExpectedOriginator;
END_METHOD

END_FUNCTION_BLOCK

// ---- mobject-collections/Tests/StackForwardEnumerator_TestSuite.TcPOU
FUNCTION_BLOCK PUBLIC StackForwardEnumerator_TestSuite EXTENDS TcUnit.FB_TestSuite

CheckIsValidAtStart();
CheckMoveNextReturnsFalseAtTheEnd();
CheckMoveNextReturnsFalseWhenEmpty();
CheckMoveNextReturnsTrueMultipleItems();
CheckMoveNextReturnsTrueSingleItem();
CheckReset();
CheckTryGet();
CheckTryGetTo();
CheckWorksWithIntegers();
CheckWorksWithStrings();
CheckWorksWithArrays();

METHOD PUBLIC CheckIsValidAtStart
VAR
	result : BOOL;
	stack : Stack;
	enumerator : I_ForwardEnumerator;
END_VAR
TEST('CheckIsValidAtStart');

enumerator := stack.GetEnumerator();

result := enumerator.IsValid;
enumerator.Dispose();

AssertTrue(
	Condition := result,
	Message := 'Method returned false'
);

TEST_FINISHED();
END_METHOD

METHOD PRIVATE CheckMoveNextReturnsFalseAtTheEnd
VAR
	in1 : INT := 123;
	result : BOOL;
	stack : Stack;
	enumerator : I_ForwardEnumerator;
END_VAR
TEST('CheckMoveNextReturnsFalseAtTheEnd');

stack.Push(in1);
enumerator := stack.GetEnumerator();

enumerator.MoveNext();
result := enumerator.MoveNext();
enumerator.Dispose();

AssertFalse(result,
    'MoveNext did not correctly signal the end of the enumeration');
	
TEST_FINISHED();
END_METHOD

METHOD PUBLIC CheckMoveNextReturnsFalseWhenEmpty
VAR
	result : BOOL;
	stack : Stack;
	enumerator : I_ForwardEnumerator;
END_VAR
TEST('CheckMoveNextReturnsFalseWhenEmpty');

enumerator := stack.GetEnumerator();

result := enumerator.MoveNext();
enumerator.Dispose();

AssertFalse(
	Condition := result,
	Message := 'MoveNext did not correctly signal the end of the enumeration'
);

TEST_FINISHED();
END_METHOD

METHOD PRIVATE CheckMoveNextReturnsTrueMultipleItems
VAR
	in1 : INT := 123;
	in2 : INT := 456;
	in3 : INT := 789;
	result : BOOL;
	stack : Stack;
	enumerator : I_ForwardEnumerator;
END_VAR
TEST('CheckMoveNextReturnsTrueMultipleItems');

stack.Push(in1);
stack.Push(in2);
stack.Push(in3);
enumerator := stack.GetEnumerator();

result := enumerator.MoveNext();
enumerator.Dispose();

AssertTrue(result, 'MoveNext did not correctly signal there were more items to follow');

TEST_FINISHED();
END_METHOD

METHOD PRIVATE CheckMoveNextReturnsTrueSingleItem
VAR
	in1 : INT := 123;
	result : BOOL;
	stack : Stack;
	enumerator : I_ForwardEnumerator;
END_VAR
TEST('CheckMoveNextReturnsTrueSingleItem');

stack.Push(in1);
enumerator := stack.GetEnumerator();

result := enumerator.MoveNext();
enumerator.Dispose();

AssertTrue(result,
    'MoveNext did not correctly signal there were more items to follow');
	
TEST_FINISHED();
END_METHOD

METHOD PUBLIC CheckReset
VAR
	in1 : ARRAY [0..1] OF REAL := [0.1,2.3];
	in2 : ARRAY [0..1] OF REAL := [1.2,3.4];
	in3 : ARRAY [0..1] OF REAL := [2.3,4.5];
	out : ARRAY [0..1] OF REAL;
	expected : ARRAY [0..1] OF REAL := [2.3,4.5];
	stack : Stack;
	enumerator : I_ForwardEnumerator;
END_VAR
TEST('CheckReset');

stack.Push(in1);
stack.Push(in2);
stack.Push(in3);

enumerator := stack.GetEnumerator();

enumerator.MoveNext();
enumerator.MoveNext();
enumerator.Reset();
enumerator.MoveNext();
enumerator.TryGet(out);

enumerator.Dispose();

AssertEquals(
	Expected := expected,
	Actual := out,
	Message := 'Did not produce the expected result'
);

TEST_FINISHED();
END_METHOD

METHOD PUBLIC CheckTryGet
VAR
	in : INT := 123;
	out : INT;
	expected : INT := 123;
	result : BOOL;
	stack : Stack;
	enumerator : I_ForwardEnumerator;
END_VAR
TEST('CheckTryGet');

stack.Push(in);
enumerator := stack.GetEnumerator();
enumerator.MoveNext();

result := enumerator.TryGet(out);
enumerator.Dispose();

AssertTrue(
	Condition := result,
	Message := 'Method returned false'
);

AssertEquals(
	Expected := expected,
	Actual := out,
	Message := 'Did not produce the expected result'
);

TEST_FINISHED();
END_METHOD

METHOD PUBLIC CheckTryGetTo
VAR
	in : INT := 123;
	out : INT;
	expected : INT := 123;
	result : BOOL;
	stack : Stack;
	enumerator : I_ForwardEnumerator;
END_VAR
TEST('CheckTryGetTo');

stack.Push(in);
enumerator := stack.GetEnumerator();
enumerator.MoveNext();

result := enumerator.TryGetTo(ADR(out),SIZEOF(out));
enumerator.Dispose();

AssertTrue(
	Condition := result,
	Message := 'Method returned false'
);

AssertEquals(
	Expected := expected,
	Actual := out,
	Message := 'Did not produce the expected result'
);

TEST_FINISHED();
END_METHOD

METHOD PUBLIC CheckWorksWithArrays
VAR
	in1 : ARRAY [0..1] OF REAL := [0.1,2.3];
	in2 : ARRAY [0..1] OF REAL := [1.2,3.4];
	in3 : ARRAY [0..1] OF REAL := [2.3,4.5];
	out1 : ARRAY [0..1] OF REAL;
	out2 : ARRAY [0..1] OF REAL;
	out3 : ARRAY [0..1] OF REAL;
	expected1 : ARRAY [0..1] OF REAL := [2.3,4.5];
	expected2 : ARRAY [0..1] OF REAL := [1.2,3.4];
	expected3 : ARRAY [0..1] OF REAL := [0.1,2.3];
	stack : Stack;
	enumerator : I_ForwardEnumerator;
END_VAR
TEST('CheckWorksWithArrays');

stack.Push(in1);
stack.Push(in2);
stack.Push(in3);

enumerator := stack.GetEnumerator();

enumerator.MoveNext();
enumerator.TryGet(out1);
enumerator.MoveNext();
enumerator.TryGet(out2);
enumerator.MoveNext();
enumerator.TryGet(out3);

enumerator.Dispose();

AssertEquals(
	Expected := expected1,
	Actual := out1,
	Message := 'Did not produce the expected 1st result'
);

AssertEquals(
	Expected := expected2,
	Actual := out2,
	Message := 'Did not produce the expected 2nd result'
);

AssertEquals(
	Expected := expected3,
	Actual := out3,
	Message := 'Did not produce the expected 3rd result'
);

TEST_FINISHED();
END_METHOD

METHOD PUBLIC CheckWorksWithIntegers
VAR
	in1 : INT := 123;
	in2 : INT := 234;
	in3 : INT := 345;
	out1 : INT;
	out2 : INT;
	out3 : INT;
	expected1 : INT := 345;
	expected2 : INT := 234;
	expected3 : INT := 123;
	stack : Stack;
	enumerator : I_ForwardEnumerator;
END_VAR
TEST('CheckWorksWithIntegers');

stack.Push(in1);
stack.Push(in2);
stack.Push(in3);

enumerator := stack.GetEnumerator();

enumerator.MoveNext();
enumerator.TryGet(out1);
enumerator.MoveNext();
enumerator.TryGet(out2);
enumerator.MoveNext();
enumerator.TryGet(out3);

enumerator.Dispose();

AssertEquals(
	Expected := expected1,
	Actual := out1,
	Message := 'Did not produce the expected 1st result'
);

AssertEquals(
	Expected := expected2,
	Actual := out2,
	Message := 'Did not produce the expected 2nd result'
);

AssertEquals(
	Expected := expected3,
	Actual := out3,
	Message := 'Did not produce the expected 3rd result'
);

TEST_FINISHED();
END_METHOD

METHOD PUBLIC CheckWorksWithStrings
VAR
	in1 : STRING := 'test1';
	in2 : STRING := 'test2';
	in3 : STRING := 'test3';
	out1 : STRING;
	out2 : STRING;
	out3 : STRING;
	expected1 : STRING := 'test3';
	expected2 : STRING := 'test2';
	expected3 : STRING := 'test1';
	stack : Stack;
	enumerator : I_ForwardEnumerator;
END_VAR
TEST('CheckWorksWithStrings');

stack.Push(in1);
stack.Push(in2);
stack.Push(in3);

enumerator := stack.GetEnumerator();

enumerator.MoveNext();
enumerator.TryGet(out1);
enumerator.MoveNext();
enumerator.TryGet(out2);
enumerator.MoveNext();
enumerator.TryGet(out3);

enumerator.Dispose();

AssertEquals(
	Expected := expected1,
	Actual := out1,
	Message := 'Did not produce the expected 1st result'
);

AssertEquals(
	Expected := expected2,
	Actual := out2,
	Message := 'Did not produce the expected 2nd result'
);

AssertEquals(
	Expected := expected3,
	Actual := out3,
	Message := 'Did not produce the expected 3rd result'
);

TEST_FINISHED();
END_METHOD

END_FUNCTION_BLOCK

// ---- mobject-converters/Tests/BOOL_TO_TestSuite.TcPOU
FUNCTION_BLOCK PUBLIC BOOL_TO_TestSuite EXTENDS TcUnit.FB_TestSuite
VAR
END_VAR

Check_BOOL_TO_BOOL_Max();
Check_BOOL_TO_BOOL_Min();
Check_BOOL_TO_BYTE_Max();
Check_BOOL_TO_BYTE_Min();
Check_BOOL_TO_WORD_Max();
Check_BOOL_TO_WORD_Min();
Check_BOOL_TO_DWORD_Max();
Check_BOOL_TO_DWORD_Min();
Check_BOOL_TO_LWORD_Max();
Check_BOOL_TO_LWORD_Min();
Check_BOOL_TO_SINT_Max();
Check_BOOL_TO_SINT_Min();
Check_BOOL_TO_INT_Max();
Check_BOOL_TO_INT_Min();
Check_BOOL_TO_DINT_Max();
Check_BOOL_TO_DINT_Min();
Check_BOOL_TO_LINT_Max();
Check_BOOL_TO_LINT_Min();
Check_BOOL_TO_USINT_Max();
Check_BOOL_TO_USINT_Min();
Check_BOOL_TO_UINT_Max();
Check_BOOL_TO_UINT_Min();
Check_BOOL_TO_UDINT_Max();
Check_BOOL_TO_UDINT_Min();
Check_BOOL_TO_ULINT_Max();
Check_BOOL_TO_ULINT_Min();
Check_BOOL_TO_REAL_Max();
Check_BOOL_TO_REAL_Min();
Check_BOOL_TO_LREAL_Max();
Check_BOOL_TO_LREAL_Min();
Check_BOOL_TO_TIME_Max();
Check_BOOL_TO_TIME_Min();
Check_BOOL_TO_TOD_Max();
Check_BOOL_TO_TOD_Min();
Check_BOOL_TO_DATE_Max();
Check_BOOL_TO_DATE_Min();
Check_BOOL_TO_DT_Max();
Check_BOOL_TO_DT_Min();
Check_BOOL_TO_STRING_Max();
Check_BOOL_TO_STRING_Min();

METHOD PUBLIC Check_BOOL_TO_BOOL_Max
VAR
	value : BOOL := DatatypeLimits.BOOL_MAX_VALUE;
	actual : BOOL;
	converted : BOOL;
	equal : BOOL;
END_VAR
TEST('Check_BOOL_TO_BOOL_Max');

// @TEST-RUN
converted := TryConvert_BOOL_TO_Destination(value, actual);
equal := actual = value;

// @TEST-ASSERT
AssertTrue(Condition := equal, Message := 'Did not convert BOOL to BOOL correctly');
AssertTrue(Condition := converted, Message := 'Did not report BOOL to BOOL conversion was successful');

TEST_FINISHED();
END_METHOD

METHOD PUBLIC Check_BOOL_TO_BOOL_Min
VAR
	value : BOOL := DatatypeLimits.BOOL_MIN_VALUE;
	actual : BOOL;
	converted : BOOL;
	equal : BOOL;
END_VAR
TEST('Check_BOOL_TO_BOOL_Min');

// @TEST-RUN
converted := TryConvert_BOOL_TO_Destination(value, actual);
equal := actual = value;

// @TEST-ASSERT
AssertTrue(Condition := equal, Message := 'Did not convert BOOL to BOOL correctly');
AssertTrue(Condition := converted, Message := 'Did not report BOOL to BOOL conversion was successful');

TEST_FINISHED();
END_METHOD

METHOD PUBLIC Check_BOOL_TO_BYTE_Max
VAR
	value : BOOL := DatatypeLimits.BOOL_MAX_VALUE;
	actual : BYTE;
	converted : BOOL;
	equal : BOOL;
END_VAR
TEST('Check_BOOL_TO_BYTE_Max');

// @TEST-RUN
converted := TryConvert_BOOL_TO_Destination(value, actual);
equal := actual = BOOL_TO_BYTE(value);

// @TEST-ASSERT
AssertTrue(Condition := equal, Message := 'Did not convert BOOL to BYTE correctly');
AssertTrue(Condition := converted, Message := 'Did not report BOOL to BYTE conversion was successful');

TEST_FINISHED();
END_METHOD

METHOD PUBLIC Check_BOOL_TO_BYTE_Min
VAR
	value : BOOL := DatatypeLimits.BOOL_MIN_VALUE;
	actual : BYTE;
	converted : BOOL;
	equal : BOOL;
END_VAR
TEST('Check_BOOL_TO_BYTE_Min');

// @TEST-RUN
converted := TryConvert_BOOL_TO_Destination(value, actual);
equal := actual = BOOL_TO_BYTE(value);

// @TEST-ASSERT
AssertTrue(Condition := equal, Message := 'Did not convert BOOL to BYTE correctly');
AssertTrue(Condition := converted, Message := 'Did not report BOOL to BYTE conversion was successful');

TEST_FINISHED();
END_METHOD

METHOD PUBLIC Check_BOOL_TO_DATE_Max
VAR
	value : BOOL := DatatypeLimits.BOOL_MAX_VALUE;
	actual : DATE;
	converted : BOOL;
	equal : BOOL;
END_VAR
TEST('Check_BOOL_TO_DATE_Max');

// @TEST-RUN
converted := TryConvert_BOOL_TO_Destination(value, actual);
equal := actual = BOOL_TO_DATE(value);

// @TEST-ASSERT
AssertTrue(Condition := equal, Message := 'Did not convert BOOL to DATE correctly');
AssertTrue(Condition := converted, Message := 'Did not report BOOL to DATE conversion was successful');

TEST_FINISHED();
END_METHOD

METHOD PUBLIC Check_BOOL_TO_DATE_Min
VAR
	value : BOOL := DatatypeLimits.BOOL_MIN_VALUE;
	actual : DATE;
	converted : BOOL;
	equal : BOOL;
END_VAR
TEST('Check_BOOL_TO_DATE_Min');

// @TEST-RUN
converted := TryConvert_BOOL_TO_Destination(value, actual);
equal := actual = BOOL_TO_DATE(value);

// @TEST-ASSERT
AssertTrue(Condition := equal, Message := 'Did not convert BOOL to DATE correctly');
AssertTrue(Condition := converted, Message := 'Did not report BOOL to DATE conversion was successful');

TEST_FINISHED();
END_METHOD

METHOD PUBLIC Check_BOOL_TO_DINT_Max
VAR
	value : BOOL := DatatypeLimits.BOOL_MAX_VALUE;
	actual : DINT;
	converted : BOOL;
	equal : BOOL;
END_VAR
TEST('Check_BOOL_TO_DINT_Max');

// @TEST-RUN
converted := TryConvert_BOOL_TO_Destination(value, actual);
equal := actual = BOOL_TO_DINT(value);

// @TEST-ASSERT
AssertTrue(Condition := equal, Message := 'Did not convert BOOL to DINT correctly');
AssertTrue(Condition := converted, Message := 'Did not report BOOL to DINT conversion was successful');

TEST_FINISHED();
END_METHOD

METHOD PUBLIC Check_BOOL_TO_DINT_Min
VAR
	value : BOOL := DatatypeLimits.BOOL_MIN_VALUE;
	actual : DINT;
	converted : BOOL;
	equal : BOOL;
END_VAR
TEST('Check_BOOL_TO_DINT_Min');

// @TEST-RUN
converted := TryConvert_BOOL_TO_Destination(value, actual);
equal := actual = BOOL_TO_DINT(value);

// @TEST-ASSERT
AssertTrue(Condition := equal, Message := 'Did not convert BOOL to DINT correctly');
AssertTrue(Condition := converted, Message := 'Did not report BOOL to DINT conversion was successful');

TEST_FINISHED();
END_METHOD

METHOD PUBLIC Check_BOOL_TO_DT_Max
VAR
	value : BOOL := DatatypeLimits.BOOL_MAX_VALUE;
	actual : DT;
	converted : BOOL;
	equal : BOOL;
END_VAR
TEST('Check_BOOL_TO_DT_Max');

// @TEST-RUN
converted := TryConvert_BOOL_TO_Destination(value, actual);
equal := actual = BOOL_TO_DT(value);

// @TEST-ASSERT
AssertTrue(Condition := equal, Message := 'Did not convert BOOL to DT correctly');
AssertTrue(Condition := converted, Message := 'Did not report BOOL to DT conversion was successful');

TEST_FINISHED();
END_METHOD

METHOD PUBLIC Check_BOOL_TO_DT_Min
VAR
	value : BOOL := DatatypeLimits.BOOL_MIN_VALUE;
	actual : DT;
	converted : BOOL;
	equal : BOOL;
END_VAR
TEST('Check_BOOL_TO_DT_Min');

// @TEST-RUN
converted := TryConvert_BOOL_TO_Destination(value, actual);
equal := actual = BOOL_TO_DT(value);

// @TEST-ASSERT
AssertTrue(Condition := equal, Message := 'Did not convert BOOL to DT correctly');
AssertTrue(Condition := converted, Message := 'Did not report BOOL to DT conversion was successful');

TEST_FINISHED();
END_METHOD

METHOD PUBLIC Check_BOOL_TO_DWORD_Max
VAR
	value : BOOL := DatatypeLimits.BOOL_MAX_VALUE;
	actual : DWORD;
	converted : BOOL;
	equal : BOOL;
END_VAR
TEST('Check_BOOL_TO_DWORD_Max');

// @TEST-RUN
converted := TryConvert_BOOL_TO_Destination(value, actual);
equal := actual = BOOL_TO_DWORD(value);

// @TEST-ASSERT
AssertTrue(Condition := equal, Message := 'Did not convert BOOL to DWORD correctly');
AssertTrue(Condition := converted, Message := 'Did not report BOOL to DWORD conversion was successful');

TEST_FINISHED();
END_METHOD

METHOD PUBLIC Check_BOOL_TO_DWORD_Min
VAR
	value : BOOL := DatatypeLimits.BOOL_MIN_VALUE;
	actual : DWORD;
	converted : BOOL;
	equal : BOOL;
END_VAR
TEST('Check_BOOL_TO_DWORD_Min');

// @TEST-RUN
converted := TryConvert_BOOL_TO_Destination(value, actual);
equal := actual = BOOL_TO_DWORD(value);

// @TEST-ASSERT
AssertTrue(Condition := equal, Message := 'Did not convert BOOL to DWORD correctly');
AssertTrue(Condition := converted, Message := 'Did not report BOOL to DWORD conversion was successful');

TEST_FINISHED();
END_METHOD

METHOD PUBLIC Check_BOOL_TO_INT_Max
VAR
	value : BOOL := DatatypeLimits.BOOL_MAX_VALUE;
	actual : INT;
	converted : BOOL;
	equal : BOOL;
END_VAR
TEST('Check_BOOL_TO_INT_Max');

// @TEST-RUN
converted := TryConvert_BOOL_TO_Destination(value, actual);
equal := actual = BOOL_TO_INT(value);

// @TEST-ASSERT
AssertTrue(Condition := equal, Message := 'Did not convert BOOL to INT correctly');
AssertTrue(Condition := converted, Message := 'Did not report BOOL to INT conversion was successful');

TEST_FINISHED();
END_METHOD

METHOD PUBLIC Check_BOOL_TO_INT_Min
VAR
	value : BOOL := DatatypeLimits.BOOL_MIN_VALUE;
	actual : INT;
	converted : BOOL;
	equal : BOOL;
END_VAR
TEST('Check_BOOL_TO_INT_Min');

// @TEST-RUN
converted := TryConvert_BOOL_TO_Destination(value, actual);
equal := actual = BOOL_TO_INT(value);

// @TEST-ASSERT
AssertTrue(Condition := equal, Message := 'Did not convert BOOL to INT correctly');
AssertTrue(Condition := converted, Message := 'Did not report BOOL to INT conversion was successful');

TEST_FINISHED();
END_METHOD

METHOD PUBLIC Check_BOOL_TO_LINT_Max
VAR
	value : BOOL := DatatypeLimits.BOOL_MAX_VALUE;
	actual : LINT;
	converted : BOOL;
	equal : BOOL;
END_VAR
TEST('Check_BOOL_TO_LINT_Max');

// @TEST-RUN
converted := TryConvert_BOOL_TO_Destination(value, actual);
equal := actual = BOOL_TO_LINT(value);

// @TEST-ASSERT
AssertTrue(Condition := equal, Message := 'Did not convert BOOL to LINT correctly');
AssertTrue(Condition := converted, Message := 'Did not report BOOL to LINT conversion was successful');

TEST_FINISHED();
END_METHOD

METHOD PUBLIC Check_BOOL_TO_LINT_Min
VAR
	value : BOOL := DatatypeLimits.BOOL_MIN_VALUE;
	actual : LINT;
	converted : BOOL;
	equal : BOOL;
END_VAR
TEST('Check_BOOL_TO_LINT_Min');

// @TEST-RUN
converted := TryConvert_BOOL_TO_Destination(value, actual);
equal := actual = BOOL_TO_LINT(value);

// @TEST-ASSERT
AssertTrue(Condition := equal, Message := 'Did not convert BOOL to LINT correctly');
AssertTrue(Condition := converted, Message := 'Did not report BOOL to LINT conversion was successful');

TEST_FINISHED();
END_METHOD

METHOD PUBLIC Check_BOOL_TO_LREAL_Max
VAR
	value : BOOL := DatatypeLimits.BOOL_MAX_VALUE;
	actual : LREAL;
	converted : BOOL;
	equal : BOOL;
END_VAR
TEST('Check_BOOL_TO_LREAL_Max');

// @TEST-RUN
converted := TryConvert_BOOL_TO_Destination(value, actual);
equal := actual = BOOL_TO_LREAL(value);

// @TEST-ASSERT
AssertTrue(Condition := equal, Message := 'Did not convert BOOL to LREAL correctly');
AssertTrue(Condition := converted, Message := 'Did not report BOOL to LREAL conversion was successful');

TEST_FINISHED();
END_METHOD

METHOD PUBLIC Check_BOOL_TO_LREAL_Min
VAR
	value : BOOL := DatatypeLimits.BOOL_MIN_VALUE;
	actual : LREAL;
	converted : BOOL;
	equal : BOOL;
END_VAR
TEST('Check_BOOL_TO_LREAL_Min');

// @TEST-RUN
converted := TryConvert_BOOL_TO_Destination(value, actual);
equal := actual = BOOL_TO_LREAL(value);

// @TEST-ASSERT
AssertTrue(Condition := equal, Message := 'Did not convert BOOL to LREAL correctly');
AssertTrue(Condition := converted, Message := 'Did not report BOOL to LREAL conversion was successful');

TEST_FINISHED();
END_METHOD

METHOD PUBLIC Check_BOOL_TO_LWORD_Max
VAR
	value : BOOL := DatatypeLimits.BOOL_MAX_VALUE;
	actual : LWORD;
	converted : BOOL;
	equal : BOOL;
END_VAR
TEST('Check_BOOL_TO_LWORD_Max');

// @TEST-RUN
converted := TryConvert_BOOL_TO_Destination(value, actual);
equal := actual = BOOL_TO_LWORD(value);

// @TEST-ASSERT
AssertTrue(Condition := equal, Message := 'Did not convert BOOL to LWORD correctly');
AssertTrue(Condition := converted, Message := 'Did not report BOOL to LWORD conversion was successful');

TEST_FINISHED();
END_METHOD

METHOD PUBLIC Check_BOOL_TO_LWORD_Min
VAR
	value : BOOL := DatatypeLimits.BOOL_MIN_VALUE;
	actual : LWORD;
	converted : BOOL;
	equal : BOOL;
END_VAR
TEST('Check_BOOL_TO_LWORD_Min');

// @TEST-RUN
converted := TryConvert_BOOL_TO_Destination(value, actual);
equal := actual = BOOL_TO_LWORD(value);

// @TEST-ASSERT
AssertTrue(Condition := equal, Message := 'Did not convert BOOL to LWORD correctly');
AssertTrue(Condition := converted, Message := 'Did not report BOOL to LWORD conversion was successful');

TEST_FINISHED();
END_METHOD

METHOD PUBLIC Check_BOOL_TO_REAL_Max
VAR
	value : BOOL := DatatypeLimits.BOOL_MAX_VALUE;
	actual : REAL;
	converted : BOOL;
	equal : BOOL;
END_VAR
TEST('Check_BOOL_TO_REAL_Max');

// @TEST-RUN
converted := TryConvert_BOOL_TO_Destination(value, actual);
equal := actual = BOOL_TO_REAL(value);

// @TEST-ASSERT
AssertTrue(Condition := equal, Message := 'Did not convert BOOL to REAL correctly');
AssertTrue(Condition := converted, Message := 'Did not report BOOL to REAL conversion was successful');

TEST_FINISHED();
END_METHOD

METHOD PUBLIC Check_BOOL_TO_REAL_Min
VAR
	value : BOOL := DatatypeLimits.BOOL_MIN_VALUE;
	actual : REAL;
	converted : BOOL;
	equal : BOOL;
END_VAR
TEST('Check_BOOL_TO_REAL_Min');

// @TEST-RUN
converted := TryConvert_BOOL_TO_Destination(value, actual);
equal := actual = BOOL_TO_REAL(value);

// @TEST-ASSERT
AssertTrue(Condition := equal, Message := 'Did not convert BOOL to REAL correctly');
AssertTrue(Condition := converted, Message := 'Did not report BOOL to REAL conversion was successful');

TEST_FINISHED();
END_METHOD

METHOD PUBLIC Check_BOOL_TO_SINT_Max
VAR
	value : BOOL := DatatypeLimits.BOOL_MAX_VALUE;
	actual : SINT;
	converted : BOOL;
	equal : BOOL;
END_VAR
TEST('Check_BOOL_TO_SINT_Max');

// @TEST-RUN
converted := TryConvert_BOOL_TO_Destination(value, actual);
equal := actual = BOOL_TO_SINT(value);

// @TEST-ASSERT
AssertTrue(Condition := equal, Message := 'Did not convert BOOL to SINT correctly');
AssertTrue(Condition := converted, Message := 'Did not report BOOL to SINT conversion was successful');

TEST_FINISHED();
END_METHOD

METHOD PUBLIC Check_BOOL_TO_SINT_Min
VAR
	value : BOOL := DatatypeLimits.BOOL_MIN_VALUE;
	actual : SINT;
	converted : BOOL;
	equal : BOOL;
END_VAR
TEST('Check_BOOL_TO_SINT_Min');

// @TEST-RUN
converted := TryConvert_BOOL_TO_Destination(value, actual);
equal := actual = BOOL_TO_SINT(value);

// @TEST-ASSERT
AssertTrue(Condition := equal, Message := 'Did not convert BOOL to SINT correctly');
AssertTrue(Condition := converted, Message := 'Did not report BOOL to SINT conversion was successful');

TEST_FINISHED();
END_METHOD

METHOD PUBLIC Check_BOOL_TO_STRING_Max
VAR
	value : BOOL := DatatypeLimits.BOOL_MAX_VALUE;
	actual : STRING;
	converted : BOOL;
	equal : BOOL;
END_VAR
TEST('Check_BOOL_TO_STRING_Max');

// @TEST-RUN
converted := TryConvert_BOOL_TO_Destination(value, actual);
equal := actual = BOOL_TO_STRING(value);

// @TEST-ASSERT
AssertTrue(Condition := equal, Message := 'Did not convert BOOL to STRING correctly');
AssertTrue(Condition := converted, Message := 'Did not report BOOL to STRING conversion was successful');

TEST_FINISHED();
END_METHOD

METHOD PUBLIC Check_BOOL_TO_STRING_Min
VAR
	value : BOOL := DatatypeLimits.BOOL_MIN_VALUE;
	actual : STRING;
	converted : BOOL;
	equal : BOOL;
END_VAR
TEST('Check_BOOL_TO_STRING_Min');

// @TEST-RUN
converted := TryConvert_BOOL_TO_Destination(value, actual);
equal := actual = BOOL_TO_STRING(value);

// @TEST-ASSERT
AssertTrue(Condition := equal, Message := 'Did not convert BOOL to STRING correctly');
AssertTrue(Condition := converted, Message := 'Did not report BOOL to STRING conversion was successful');

TEST_FINISHED();
END_METHOD

METHOD PUBLIC Check_BOOL_TO_TIME_Max
VAR
	value : BOOL := DatatypeLimits.BOOL_MAX_VALUE;
	actual : TIME;
	converted : BOOL;
	equal : BOOL;
END_VAR
TEST('Check_BOOL_TO_TIME_Max');

// @TEST-RUN
converted := TryConvert_BOOL_TO_Destination(value, actual);
equal := actual = BOOL_TO_TIME(value);

// @TEST-ASSERT
AssertTrue(Condition := equal, Message := 'Did not convert BOOL to TIME correctly');
AssertTrue(Condition := converted, Message := 'Did not report BOOL to TIME conversion was successful');

TEST_FINISHED();
END_METHOD

METHOD PUBLIC Check_BOOL_TO_TIME_Min
VAR
	value : BOOL := DatatypeLimits.BOOL_MIN_VALUE;
	actual : TIME;
	converted : BOOL;
	equal : BOOL;
END_VAR
TEST('Check_BOOL_TO_TIME_Min');

// @TEST-RUN
converted := TryConvert_BOOL_TO_Destination(value, actual);
equal := actual = BOOL_TO_TIME(value);

// @TEST-ASSERT
AssertTrue(Condition := equal, Message := 'Did not convert BOOL to TIME correctly');
AssertTrue(Condition := converted, Message := 'Did not report BOOL to TIME conversion was successful');

TEST_FINISHED();
END_METHOD

METHOD PUBLIC Check_BOOL_TO_TOD_Max
VAR
	value : BOOL := DatatypeLimits.BOOL_MAX_VALUE;
	actual : TOD;
	converted : BOOL;
	equal : BOOL;
END_VAR
TEST('Check_BOOL_TO_TOD_Max');

// @TEST-RUN
converted := TryConvert_BOOL_TO_Destination(value, actual);
equal := actual = BOOL_TO_TOD(value);

// @TEST-ASSERT
AssertTrue(Condition := equal, Message := 'Did not convert BOOL to TOD correctly');
AssertTrue(Condition := converted, Message := 'Did not report BOOL to TOD conversion was successful');

TEST_FINISHED();
END_METHOD

METHOD PUBLIC Check_BOOL_TO_TOD_Min
VAR
	value : BOOL := DatatypeLimits.BOOL_MIN_VALUE;
	actual : TOD;
	converted : BOOL;
	equal : BOOL;
END_VAR
TEST('Check_BOOL_TO_TOD_Min');

// @TEST-RUN
converted := TryConvert_BOOL_TO_Destination(value, actual);
equal := actual = BOOL_TO_TOD(value);

// @TEST-ASSERT
AssertTrue(Condition := equal, Message := 'Did not convert BOOL to TOD correctly');
AssertTrue(Condition := converted, Message := 'Did not report BOOL to TOD conversion was successful');

TEST_FINISHED();
END_METHOD

METHOD PUBLIC Check_BOOL_TO_UDINT_Max
VAR
	value : BOOL := DatatypeLimits.BOOL_MAX_VALUE;
	actual : UDINT;
	converted : BOOL;
	equal : BOOL;
END_VAR
TEST('Check_BOOL_TO_UDINT_Max');

// @TEST-RUN
converted := TryConvert_BOOL_TO_Destination(value, actual);
equal := actual = BOOL_TO_UDINT(value);

// @TEST-ASSERT
AssertTrue(Condition := equal, Message := 'Did not convert BOOL to UDINT correctly');
AssertTrue(Condition := converted, Message := 'Did not report BOOL to UDINT conversion was successful');

TEST_FINISHED();
END_METHOD

METHOD PUBLIC Check_BOOL_TO_UDINT_Min
VAR
	value : BOOL := DatatypeLimits.BOOL_MIN_VALUE;
	actual : UDINT;
	converted : BOOL;
	equal : BOOL;
END_VAR
TEST('Check_BOOL_TO_UDINT_Min');

// @TEST-RUN
converted := TryConvert_BOOL_TO_Destination(value, actual);
equal := actual = BOOL_TO_UDINT(value);

// @TEST-ASSERT
AssertTrue(Condition := equal, Message := 'Did not convert BOOL to UDINT correctly');
AssertTrue(Condition := converted, Message := 'Did not report BOOL to UDINT conversion was successful');

TEST_FINISHED();
END_METHOD

METHOD PUBLIC Check_BOOL_TO_UINT_Max
VAR
	value : BOOL := DatatypeLimits.BOOL_MAX_VALUE;
	actual : UINT;
	converted : BOOL;
	equal : BOOL;
END_VAR
TEST('Check_BOOL_TO_UINT_Max');

// @TEST-RUN
converted := TryConvert_BOOL_TO_Destination(value, actual);
equal := actual = BOOL_TO_UINT(value);

// @TEST-ASSERT
AssertTrue(Condition := equal, Message := 'Did not convert BOOL to UINT correctly');
AssertTrue(Condition := converted, Message := 'Did not report BOOL to UINT conversion was successful');

TEST_FINISHED();
END_METHOD

METHOD PUBLIC Check_BOOL_TO_UINT_Min
VAR
	value : BOOL := DatatypeLimits.BOOL_MIN_VALUE;
	actual : UINT;
	converted : BOOL;
	equal : BOOL;
END_VAR
TEST('Check_BOOL_TO_UINT_Min');

// @TEST-RUN
converted := TryConvert_BOOL_TO_Destination(value, actual);
equal := actual = BOOL_TO_UINT(value);

// @TEST-ASSERT
AssertTrue(Condition := equal, Message := 'Did not convert BOOL to UINT correctly');
AssertTrue(Condition := converted, Message := 'Did not report BOOL to UINT conversion was successful');

TEST_FINISHED();
END_METHOD

METHOD PUBLIC Check_BOOL_TO_ULINT_Max
VAR
	value : BOOL := DatatypeLimits.BOOL_MAX_VALUE;
	actual : ULINT;
	converted : BOOL;
	equal : BOOL;
END_VAR
TEST('Check_BOOL_TO_ULINT_Max');

// @TEST-RUN
converted := TryConvert_BOOL_TO_Destination(value, actual);
equal := actual = BOOL_TO_ULINT(value);

// @TEST-ASSERT
AssertTrue(Condition := equal, Message := 'Did not convert BOOL to ULINT correctly');
AssertTrue(Condition := converted, Message := 'Did not report BOOL to ULINT conversion was successful');

TEST_FINISHED();
END_METHOD

METHOD PUBLIC Check_BOOL_TO_ULINT_Min
VAR
	value : BOOL := DatatypeLimits.BOOL_MIN_VALUE;
	actual : ULINT;
	converted : BOOL;
	equal : BOOL;
END_VAR
TEST('Check_BOOL_TO_ULINT_Min');

// @TEST-RUN
converted := TryConvert_BOOL_TO_Destination(value, actual);
equal := actual = BOOL_TO_ULINT(value);

// @TEST-ASSERT
AssertTrue(Condition := equal, Message := 'Did not convert BOOL to ULINT correctly');
AssertTrue(Condition := converted, Message := 'Did not report BOOL to ULINT conversion was successful');

TEST_FINISHED();
END_METHOD

METHOD PUBLIC Check_BOOL_TO_USINT_Max
VAR
	value : BOOL := DatatypeLimits.BOOL_MAX_VALUE;
	actual : USINT;
	converted : BOOL;
	equal : BOOL;
END_VAR
TEST('Check_BOOL_TO_USINT_Max');

// @TEST-RUN
converted := TryConvert_BOOL_TO_Destination(value, actual);
equal := actual = BOOL_TO_USINT(value);

// @TEST-ASSERT
AssertTrue(Condition := equal, Message := 'Did not convert BOOL to USINT correctly');
AssertTrue(Condition := converted, Message := 'Did not report BOOL to USINT conversion was successful');

TEST_FINISHED();
END_METHOD

METHOD PUBLIC Check_BOOL_TO_USINT_Min
VAR
	value : BOOL := DatatypeLimits.BOOL_MIN_VALUE;
	actual : USINT;
	converted : BOOL;
	equal : BOOL;
END_VAR
TEST('Check_BOOL_TO_USINT_Min');

// @TEST-RUN
converted := TryConvert_BOOL_TO_Destination(value, actual);
equal := actual = BOOL_TO_USINT(value);

// @TEST-ASSERT
AssertTrue(Condition := equal, Message := 'Did not convert BOOL to USINT correctly');
AssertTrue(Condition := converted, Message := 'Did not report BOOL to USINT conversion was successful');

TEST_FINISHED();
END_METHOD

METHOD PUBLIC Check_BOOL_TO_WORD_Max
VAR
	value : BOOL := DatatypeLimits.BOOL_MAX_VALUE;
	actual : WORD;
	converted : BOOL;
	equal : BOOL;
END_VAR
TEST('Check_BOOL_TO_WORD_Max');

// @TEST-RUN
converted := TryConvert_BOOL_TO_Destination(value, actual);
equal := actual = BOOL_TO_WORD(value);

// @TEST-ASSERT
AssertTrue(Condition := equal, Message := 'Did not convert BOOL to WORD correctly');
AssertTrue(Condition := converted, Message := 'Did not report BOOL to WORD conversion was successful');

TEST_FINISHED();
END_METHOD

METHOD PUBLIC Check_BOOL_TO_WORD_Min
VAR
	value : BOOL := DatatypeLimits.BOOL_MIN_VALUE;
	actual : WORD;
	converted : BOOL;
	equal : BOOL;
END_VAR
TEST('Check_BOOL_TO_WORD_Min');

// @TEST-RUN
converted := TryConvert_BOOL_TO_Destination(value, actual);
equal := actual = BOOL_TO_WORD(value);

// @TEST-ASSERT
AssertTrue(Condition := equal, Message := 'Did not convert BOOL to WORD correctly');
AssertTrue(Condition := converted, Message := 'Did not report BOOL to WORD conversion was successful');

TEST_FINISHED();
END_METHOD

END_FUNCTION_BLOCK

// ---- mobject-converters/Tests/DT_TO_TestSuite.TcPOU
FUNCTION_BLOCK PUBLIC DT_TO_TestSuite EXTENDS TcUnit.FB_TestSuite
VAR
END_VAR

Check_DT_TO_BOOL_Max();
Check_DT_TO_BOOL_Min();
Check_DT_TO_BYTE_Max();
Check_DT_TO_BYTE_Min();
Check_DT_TO_BYTE_TooHigh();
Check_DT_TO_WORD_Max();
Check_DT_TO_WORD_Min();
Check_DT_TO_WORD_TooHigh();
Check_DT_TO_DWORD_Max();
Check_DT_TO_DWORD_Min();
Check_DT_TO_LWORD_Max();
Check_DT_TO_LWORD_Min();
Check_DT_TO_SINT_Max();
Check_DT_TO_SINT_Min();
Check_DT_TO_SINT_TooHigh();
Check_DT_TO_INT_Max();
Check_DT_TO_INT_Min();
Check_DT_TO_INT_TooHigh();
Check_DT_TO_DINT_Max();
Check_DT_TO_DINT_Min();
Check_DT_TO_DINT_TooHigh();
Check_DT_TO_LINT_Max();
Check_DT_TO_LINT_Min();
Check_DT_TO_USINT_Max();
Check_DT_TO_USINT_Min();
Check_DT_TO_USINT_TooHigh();
Check_DT_TO_UINT_Max();
Check_DT_TO_UINT_Min();
Check_DT_TO_UINT_TooHigh();
Check_DT_TO_UDINT_Max();
Check_DT_TO_UDINT_Min();
Check_DT_TO_ULINT_Max();
Check_DT_TO_ULINT_Min();
Check_DT_TO_REAL_Max();
Check_DT_TO_REAL_Min();
Check_DT_TO_LREAL_Max();
Check_DT_TO_LREAL_Min();
Check_DT_TO_TIME_Max();
Check_DT_TO_TIME_Min();
Check_DT_TO_TIME_TooHigh();
Check_DT_TO_TOD_Max();
Check_DT_TO_TOD_Min();
Check_DT_TO_TOD_TooHigh();
Check_DT_TO_DATE_Max();
Check_DT_TO_DATE_Min();
Check_DT_TO_DT_Max();
Check_DT_TO_DT_Min();
Check_DT_TO_STRING_Max();
Check_DT_TO_STRING_Min();

METHOD PUBLIC Check_DT_TO_BOOL_Max
VAR
	value : DT := DatatypeLimits.DT_MAX_VALUE;
	actual : BOOL;
	converted : BOOL;
	equal : BOOL;
END_VAR
TEST('Check_DT_TO_BOOL_Max');

// @TEST-RUN
converted := TryConvert_DT_TO_Destination(value, actual);
equal := actual = DT_TO_BOOL(value);

// @TEST-ASSERT
AssertTrue(Condition := equal, Message := 'Did not convert DT to BOOL correctly');
AssertTrue(Condition := converted, Message := 'Did not report DT to BOOL conversion was successful');

TEST_FINISHED();
END_METHOD

METHOD PUBLIC Check_DT_TO_BOOL_Min
VAR
	value : DT := DatatypeLimits.DT_MIN_VALUE;
	actual : BOOL;
	converted : BOOL;
	equal : BOOL;
END_VAR
TEST('Check_DT_TO_BOOL_Min');

// @TEST-RUN
converted := TryConvert_DT_TO_Destination(value, actual);
equal := actual = DT_TO_BOOL(value);

// @TEST-ASSERT
AssertTrue(Condition := equal, Message := 'Did not convert DT to BOOL correctly');
AssertTrue(Condition := converted, Message := 'Did not report DT to BOOL conversion was successful');

TEST_FINISHED();
END_METHOD

METHOD PUBLIC Check_DT_TO_BYTE_Max
VAR
	value : DT := DatatypeLimits.MAX_VALUE_OF_DT_WHICH_CAN_BE_HELD_IN_A_BYTE;
	actual : BYTE;
	converted : BOOL;
	equal : BOOL;
END_VAR
TEST('Check_DT_TO_BYTE_Max');

// @TEST-RUN
converted := TryConvert_DT_TO_Destination(value, actual);
equal := actual = DT_TO_BYTE(value);

// @TEST-ASSERT
AssertTrue(Condition := equal, Message := 'Did not convert DT to BYTE correctly');
AssertTrue(Condition := converted, Message := 'Did not report DT to BYTE conversion was successful');

TEST_FINISHED();
END_METHOD

METHOD PUBLIC Check_DT_TO_BYTE_Min
VAR
	value : DT := DatatypeLimits.DT_MIN_VALUE;
	actual : BYTE;
	converted : BOOL;
	equal : BOOL;
END_VAR
TEST('Check_DT_TO_BYTE_Min');

// @TEST-RUN
converted := TryConvert_DT_TO_Destination(value, actual);
equal := actual = DT_TO_BYTE(value);

// @TEST-ASSERT
AssertTrue(Condition := equal, Message := 'Did not convert DT to BYTE correctly');
AssertTrue(Condition := converted, Message := 'Did not report DT to BYTE conversion was successful');

TEST_FINISHED();
END_METHOD

METHOD PUBLIC Check_DT_TO_BYTE_TooHigh
VAR
	value : DT := DatatypeLimits.DT_MAX_VALUE;
	actual : BYTE;
	converted : BOOL;
END_VAR
TEST('Check_DT_TO_BYTE_TooHigh');

// @TEST-RUN
converted := TryConvert_DT_TO_Destination(value, actual);

// @TEST-ASSERT
AssertFalse(Condition := converted, Message := 'Did not report DT to BYTE conversion was prevented');

TEST_FINISHED();
END_METHOD

METHOD PUBLIC Check_DT_TO_DATE_Max
VAR
	value : DT := DatatypeLimits.DT_MAX_VALUE;
	actual : DATE;
	converted : BOOL;
	equal : BOOL;
END_VAR
TEST('Check_DT_TO_DATE_Max');

// @TEST-RUN
converted := TryConvert_DT_TO_Destination(value, actual);
equal := actual = DT_TO_DATE(value);

// @TEST-ASSERT
AssertTrue(Condition := equal, Message := 'Did not convert DT to DATE correctly');
AssertTrue(Condition := converted, Message := 'Did not report DT to DATE conversion was successful');

TEST_FINISHED();
END_METHOD

METHOD PUBLIC Check_DT_TO_DATE_Min
VAR
	value : DT := DatatypeLimits.DT_MIN_VALUE;
	actual : DATE;
	converted : BOOL;
	equal : BOOL;
END_VAR
TEST('Check_DT_TO_DATE_Min');

// @TEST-RUN
converted := TryConvert_DT_TO_Destination(value, actual);
equal := actual = DT_TO_DATE(value);

// @TEST-ASSERT
AssertTrue(Condition := equal, Message := 'Did not convert DT to DATE correctly');
AssertTrue(Condition := converted, Message := 'Did not report DT to DATE conversion was successful');

TEST_FINISHED();
END_METHOD

